Yaskawa INFORM job: BATMAN_NEW3.JBI

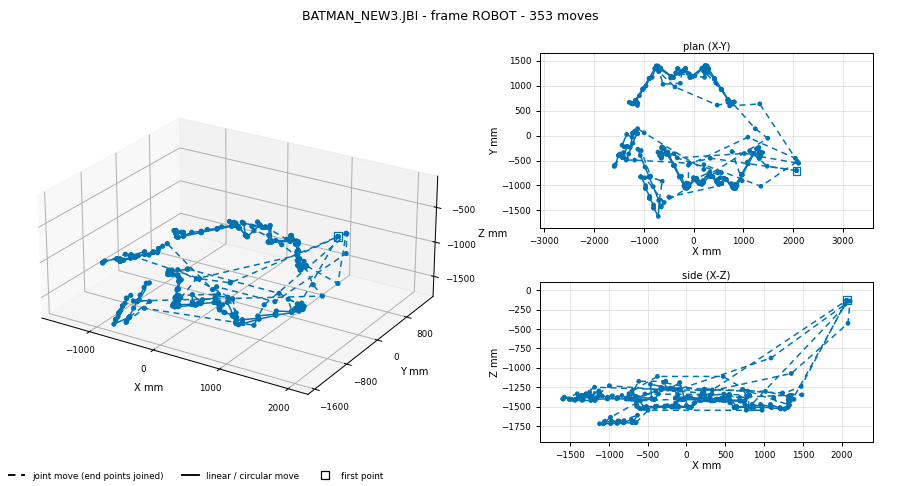
[picture p0: tool path of BATMAN_NEW3.JBI in frame ROBOT, 353 of 354 moves have a stored position in this frame; points joined in program order, loops and branches not executed]
/JOB
//NAME BATMAN_NEW3
//POS
///NPOS 437,437,353,19,0,1
///TOOL 0
///POSTYPE ROBOT
///RECTAN
///RCONF 0,0,0,0,0,0,0,0,0,0,0,0,0,0,0,0,0,0,0,0,0,0,0,0
C00000=2065.993,-701.065,-130.284,1.6748,-19.7957,-6.8086
C00001=2065.993,-701.066,-130.317,1.6736,-19.7947,-6.8065
C00002=1479.209,-614.254,-1239.827,11.6326,33.9671,-178.8219
C00003=1125.636,-307.051,-1381.425,11.6326,33.9683,179.6301
C00004=1211.356,-355.995,-1515.705,1.6711,33.5119,145.1887
C00005=1207.829,-356.009,-1519.032,1.6708,33.5119,145.1897
C00006=1207.807,-355.998,-1529.580,1.6710,33.5101,145.1899
C00007=1207.829,-356.009,-1519.032,1.6708,33.5119,145.1897
C00008=1226.216,-355.997,-1519.056,1.6724,33.5092,145.1902
C00009=1207.829,-356.009,-1519.032,1.6708,33.5119,145.1897
C00010=1082.252,-529.394,-1470.919,1.6706,33.5110,145.1945
C00011=1087.987,-562.193,-1501.828,1.6729,33.5117,145.1983
C00012=1088.014,-562.206,-1515.111,1.6726,33.5132,145.1983
C00013=1087.987,-562.193,-1501.828,1.6729,33.5117,145.1983
C00014=1116.737,-562.190,-1501.837,1.6716,33.5119,145.1949
C00015=1087.987,-562.193,-1501.828,1.6729,33.5117,145.1983
C00016=956.028,-780.276,-1470.920,1.6694,33.5121,145.1915
C00017=968.960,-788.125,-1498.527,1.6701,33.5115,145.1891
C00018=968.967,-788.120,-1508.943,1.6694,33.5115,145.1892
C00019=968.960,-788.125,-1498.527,1.6701,33.5115,145.1891
C00020=991.209,-788.123,-1498.543,1.6717,33.5108,145.1905
C00021=968.960,-788.125,-1498.527,1.6701,33.5115,145.1891
C00022=846.889,-978.207,-1470.921,1.6701,33.5116,145.1891
C00023=862.357,-1002.638,-1501.051,1.6670,33.5088,145.1850
C00024=862.345,-1002.624,-1509.122,1.6663,33.5074,145.1836
C00025=862.357,-1002.638,-1501.051,1.6670,33.5088,145.1850
C00026=878.170,-1002.616,-1501.076,1.6660,33.5090,145.1863
C00027=862.357,-1002.638,-1501.051,1.6670,33.5088,145.1850
C00028=751.878,-962.551,-1470.637,-9.9278,21.9341,47.3593
C00029=782.343,-1021.883,-1501.453,-6.5198,31.4589,38.6711
C00030=782.349,-1021.901,-1508.593,-6.5211,31.4595,38.6707
C00031=782.343,-1021.883,-1501.453,-6.5198,31.4589,38.6711
C00032=772.436,-1031.632,-1503.007,-6.5210,31.4603,38.6751
C00033=782.343,-1021.883,-1501.453,-6.5198,31.4589,38.6711
C00034=651.465,-878.509,-1502.529,-6.5193,31.4567,38.6726
C00035=649.681,-879.962,-1505.034,-6.5204,31.4570,38.6688
C00036=649.679,-879.971,-1512.967,-6.5216,31.4579,38.6721
C00037=649.681,-879.962,-1505.034,-6.5204,31.4570,38.6688
C00038=638.496,-885.487,-1507.904,-6.5213,31.4572,38.6690
C00039=649.681,-879.962,-1505.034,-6.5204,31.4570,38.6688
C00040=536.093,-844.110,-1358.224,-6.5194,31.4565,38.6698
C00041=485.208,-882.506,-1390.226,-6.5180,31.4566,38.6722
C00042=469.831,-925.588,-1412.310,-6.5196,31.4595,38.6720
C00043=469.838,-925.615,-1422.209,-6.5208,31.4607,38.6737
C00044=469.831,-925.588,-1412.310,-6.5196,31.4595,38.6720
C00045=460.916,-939.180,-1415.903,-6.5217,31.4610,38.6723
C00046=469.831,-925.588,-1412.310,-6.5196,31.4595,38.6720
C00047=390.944,-821.413,-1401.907,-6.5189,31.4593,38.6711
C00048=370.304,-823.702,-1415.949,-6.5184,31.4594,38.6679
C00049=370.309,-823.695,-1427.366,-6.5174,31.4589,38.6696
C00050=370.304,-823.702,-1415.949,-6.5184,31.4594,38.6679
C00051=362.481,-832.843,-1419.419,-6.5181,31.4591,38.6684
C00052=370.304,-823.702,-1415.949,-6.5184,31.4594,38.6679
C00053=304.377,-775.536,-1384.314,-6.5183,31.4594,38.6652
C00054=190.919,-901.974,-1384.308,6.6118,30.8401,128.8238
C00055=195.878,-934.762,-1411.685,6.6092,30.8405,128.8212
C00056=195.887,-934.767,-1420.325,6.6101,30.8407,128.8263
C00057=195.878,-934.762,-1411.685,6.6092,30.8405,128.8212
C00058=202.495,-948.084,-1414.851,6.6099,30.8403,128.8223
C00059=195.878,-934.762,-1411.685,6.6092,30.8405,128.8212
C00060=-1.386,-846.899,-1381.133,6.6069,30.8405,134.1399
C00061=-1.384,-846.902,-1485.292,6.6071,30.8406,134.1408
C00062=18.120,-884.199,-1503.049,6.6086,30.8410,134.1399
C00063=18.115,-884.194,-1511.506,6.6087,30.8409,134.1387
C00064=18.120,-884.199,-1503.049,6.6086,30.8410,134.1399
C00065=26.172,-895.008,-1505.663,6.6092,30.8415,134.1385
C00066=18.120,-884.199,-1503.049,6.6086,30.8410,134.1399
C00067=-111.813,-1001.782,-1489.786,6.6089,30.8396,134.1409
C00068=-110.516,-1020.985,-1499.218,6.6089,30.8402,134.1417
C00069=-110.523,-1020.998,-1507.131,6.6095,30.8409,134.1397
C00070=-110.516,-1020.985,-1499.218,6.6089,30.8402,134.1417
C00071=-104.498,-1031.543,-1502.310,6.6099,30.8394,134.1431
C00072=-110.516,-1020.985,-1499.218,6.6089,30.8402,134.1417
C00073=-134.961,-974.431,-1451.204,-0.2767,36.0814,31.9882
C00074=-184.395,-1006.620,-1494.709,-0.2788,36.0816,31.9875
C00075=-184.386,-1006.637,-1507.407,-0.2801,36.0816,31.9874
C00076=-184.395,-1006.620,-1494.709,-0.2788,36.0816,31.9875
C00077=-208.747,-1006.634,-1494.698,-0.2814,36.0810,31.9855
C00078=-184.395,-1006.620,-1494.709,-0.2788,36.0816,31.9875
C00079=-244.393,-814.940,-1486.725,-0.2795,36.0814,31.9846
C00080=-276.066,-822.621,-1495.047,-0.2812,36.0816,31.9820
C00081=-276.076,-822.621,-1505.407,-0.2803,36.0821,31.9829
C00082=-276.066,-822.621,-1495.047,-0.2812,36.0816,31.9820
C00083=-299.433,-822.605,-1495.065,-0.2798,36.0806,31.9846
C00084=-276.066,-822.621,-1495.047,-0.2812,36.0816,31.9820
C00085=-381.996,-597.063,-1495.018,-0.2830,36.0831,31.9834
C00086=-396.395,-597.055,-1498.231,-0.2823,36.0831,31.9838
C00087=-396.413,-597.067,-1510.313,-0.2821,36.0844,31.9835
C00088=-396.395,-597.055,-1498.231,-0.2823,36.0831,31.9838
C00089=-422.077,-597.035,-1498.242,-0.2815,36.0825,31.9834
C00090=-396.395,-597.055,-1498.231,-0.2823,36.0831,31.9838
C00091=-516.342,-329.683,-1498.242,-0.2858,36.0793,31.9791
C00092=-541.396,-335.433,-1515.036,-0.2853,36.0793,31.9798
C00093=-541.399,-335.427,-1525.902,-0.2848,36.0790,31.9796
C00094=-541.396,-335.433,-1515.036,-0.2853,36.0793,31.9798
C00095=-563.435,-335.446,-1515.016,-0.2858,36.0816,31.9782
C00096=-541.396,-335.433,-1515.036,-0.2853,36.0793,31.9798
C00097=-641.458,-364.123,-1372.142,-0.2839,36.0778,31.9819
C00098=-662.744,-397.701,-1394.268,-0.2832,36.0779,31.9810
C00099=-662.752,-397.694,-1404.858,-0.2824,36.0779,31.9809
C00100=-662.744,-397.701,-1394.268,-0.2832,36.0779,31.9810
C00101=-686.425,-397.683,-1394.265,-0.2810,36.0766,31.9839
C00102=-662.744,-397.701,-1394.268,-0.2832,36.0779,31.9810
C00103=-395.220,-362.676,-1299.812,-0.2837,36.0781,31.9812
C00104=-328.978,-445.538,-1251.827,-0.2820,36.0777,31.9846
C00105=1019.066,-358.271,-1303.588,-0.7093,36.3388,173.5111
C00106=1312.502,-388.638,-1368.088,-0.7090,36.3391,143.8761
C00107=1330.261,-409.263,-1395.611,-0.7097,36.3382,143.8752
C00108=1330.266,-409.258,-1408.665,-0.7105,36.3381,143.8742
C00109=1330.261,-409.263,-1395.611,-0.7097,36.3382,143.8752
C00110=1359.166,-409.282,-1395.624,-0.7081,36.3381,143.8755
C00111=1330.261,-409.263,-1395.611,-0.7097,36.3382,143.8752
C00112=1346.256,-330.236,-1377.208,-0.7085,36.3387,143.8760
C00113=1385.768,-339.505,-1405.683,-0.7074,36.3385,143.8819
C00114=1349.259,-407.967,-1405.698,-0.7099,36.3376,143.8723
C00115=1344.221,-409.875,-1407.374,-0.7109,36.3390,143.8722
C00116=1319.007,-459.412,-1408.358,-0.7127,36.3385,143.8707
C00117=1316.585,-457.113,-1411.355,-0.7151,36.3388,143.8640
C00118=1314.211,-431.828,-1419.878,-0.7170,36.3383,163.2059
C00119=1313.610,-343.846,-1457.563,-0.7163,36.3370,163.2057
C00120=1312.128,-239.426,-1504.329,-0.7192,36.3404,-169.8403
C00121=1302.531,-244.407,-1511.260,-0.7169,36.3409,-169.8377
C00122=1267.911,-263.148,-1529.181,-0.7174,36.3418,-169.8424
C00123=1265.622,-266.346,-1531.847,1.6688,33.5119,174.0846
C00124=1213.936,-359.434,-1529.128,7.9444,32.4168,142.7983
C00125=1097.826,-565.399,-1513.792,8.0761,31.8062,143.0840
C00126=978.992,-787.849,-1508.370,11.5262,32.2738,144.8308
C00127=870.875,-1002.933,-1509.595,7.8980,31.3909,142.8673
C00128=841.816,-1062.860,-1508.469,7.3802,28.2390,142.8982
C00129=553.926,-745.251,-1344.470,9.9580,22.3671,144.0884
C00130=553.926,-745.251,-1344.470,9.9580,22.3671,144.0884
C00131=-536.407,-379.228,-1337.930,-3.7346,30.6001,32.3556
C00132=-716.129,-331.806,-1403.803,-3.7368,30.5972,32.3471
C00133=-681.265,-398.771,-1403.765,-3.7327,30.5994,32.3525
C00134=-676.698,-399.723,-1405.572,-3.7330,30.6001,32.3555
C00135=-648.225,-452.003,-1403.979,-3.7329,30.5991,32.3574
C00136=-645.783,-446.417,-1409.426,-3.7316,30.5985,32.3594
C00137=-643.641,-424.031,-1414.162,6.8151,41.7178,38.5590
C00138=-642.472,-351.082,-1444.628,6.8142,41.7174,38.5597
C00139=-641.451,-256.638,-1485.774,6.7766,41.4625,22.9438
C00140=-638.655,-225.961,-1497.533,6.8201,41.7201,-9.7951
C00141=-606.472,-247.507,-1518.640,6.8237,41.7199,-9.7921
C00142=-589.700,-266.409,-1527.585,-3.7338,30.5952,1.6448
C00143=-548.411,-343.534,-1525.056,-3.7347,30.5964,37.9422
C00144=-403.963,-602.728,-1509.074,-3.7352,30.6012,40.7690
C00145=-284.220,-831.531,-1505.467,-3.7335,30.6016,39.5000
C00146=-193.310,-1012.463,-1505.473,-3.7341,30.5995,40.3635
C00147=-172.149,-1053.927,-1503.363,-3.7384,30.5988,41.1995
C00148=-143.820,-951.201,-1386.733,-3.7395,30.5979,32.3557
C00149=328.849,-733.445,-1337.611,2.7644,30.8890,70.6747
C00150=338.434,-799.747,-1424.588,2.7649,30.8868,70.6709
C00151=347.582,-809.529,-1424.840,2.7655,30.8869,70.6739
C00152=465.382,-936.963,-1420.390,2.7641,30.8894,70.6728
C00153=500.403,-974.854,-1419.495,2.7654,30.8881,70.6755
C00154=502.728,-975.948,-1420.152,2.7642,30.8887,70.6768
C00155=558.235,-964.171,-1445.639,29.9134,35.7054,85.7902
C00156=566.476,-953.294,-1452.395,19.5078,42.2162,79.2507
C00157=613.155,-854.018,-1511.422,19.5140,42.2128,79.2557
C00158=619.425,-859.852,-1512.190,3.7143,38.7707,68.9580
C00159=645.641,-886.484,-1510.742,-0.5875,30.5403,66.8343
C00160=773.682,-1027.269,-1508.152,1.6003,33.1198,67.9708
C00161=802.111,-1056.994,-1506.134,3.6680,32.7298,69.0087
C00162=802.122,-1056.982,-1354.174,6.2530,30.6739,70.3394
C00163=481.154,-746.898,-1337.541,6.2536,30.6743,70.3404
C00164=303.930,-769.190,-1354.154,12.5353,29.0330,117.3688
C00165=330.093,-802.167,-1423.714,12.5353,29.0320,117.3702
C00166=314.789,-820.264,-1426.190,12.5335,29.0340,117.3719
C00167=194.430,-949.182,-1419.608,12.5356,29.0341,117.3712
C00168=168.116,-977.659,-1418.609,12.5346,29.0295,117.3793
C00169=164.056,-975.884,-1418.609,12.5348,29.0312,117.3768
C00170=109.552,-964.850,-1447.287,-20.8943,38.2908,98.4122
C00171=97.137,-940.053,-1460.340,-8.8476,43.5866,106.1670
C00172=64.741,-867.815,-1502.677,-8.8482,43.5869,106.1635
C00173=57.160,-853.414,-1511.897,-8.8466,43.5860,106.1711
C00174=48.710,-862.514,-1512.138,-8.7696,29.7613,106.6801
C00175=-100.586,-1023.322,-1507.723,-8.7691,29.7615,106.6747
C00176=-133.949,-1058.932,-1505.596,-8.7707,29.7582,106.6747
C00177=-104.193,-961.904,-1408.358,-8.7704,29.7603,106.6778
C00178=-104.195,-589.697,-1279.272,-8.7711,29.7586,106.6768
C00179=1089.919,-31.439,-873.125,-36.7541,69.9873,137.0084
///RCONF 0,0,0,0,1,0,0,0,0,0,0,0,0,0,0,0,0,0,0,0,0,0,0,0
C00180=2042.728,-454.958,-183.433,1.6788,-19.8065,-6.7510
C00181=1329.047,637.602,-1479.857,8.0540,25.5528,30.8439
///RCONF 0,0,0,0,0,0,0,0,0,0,0,0,0,0,0,0,0,0,0,0,0,0,0,0
C00182=724.107,597.545,-1276.344,-3.2635,41.6684,-140.4024
C00183=785.383,659.459,-1372.820,-3.2632,41.6678,-140.4000
C00184=792.753,652.576,-1383.361,-3.2644,41.6697,-140.4060
C00185=785.383,659.459,-1372.820,-3.2632,41.6678,-140.4000
C00186=780.124,673.327,-1385.992,-3.2593,41.6675,-140.3923
C00187=785.383,659.459,-1372.820,-3.2632,41.6678,-140.4000
C00188=688.781,670.593,-1383.775,8.5921,32.7651,-134.9169
C00189=689.238,716.401,-1420.123,8.5921,32.7651,-134.9151
C00190=689.245,716.402,-1430.226,8.5926,32.7655,-134.9147
C00191=689.238,716.401,-1420.123,8.5921,32.7651,-134.9151
C00192=710.026,716.388,-1420.124,8.5932,32.7632,-134.9113
C00193=689.238,716.401,-1420.123,8.5921,32.7651,-134.9151
C00194=689.230,716.407,-1420.121,8.5916,32.7651,-134.9153
C00195=554.239,927.574,-1413.741,8.5900,32.7633,-134.9152
C00196=554.238,927.566,-1425.025,8.5905,32.7628,-134.9151
C00197=554.239,927.574,-1413.741,8.5900,32.7633,-134.9152
C00198=579.309,927.583,-1413.727,8.5909,32.7646,-134.9144
C00199=554.239,927.574,-1413.741,8.5900,32.7633,-134.9152
C00200=447.851,1057.003,-1392.108,8.5896,32.7630,-134.9175
C00201=417.599,1139.232,-1408.122,8.5926,32.7611,-134.9068
C00202=417.620,1139.241,-1415.890,8.5939,32.7624,-134.9057
C00203=417.599,1139.232,-1408.122,8.5926,32.7611,-134.9068
C00204=437.176,1139.232,-1408.121,8.5924,32.7608,-134.9064
C00205=417.599,1139.232,-1408.122,8.5926,32.7611,-134.9068
C00206=298.416,1271.074,-1391.633,8.5930,32.7623,-134.9078
C00207=293.017,1340.342,-1403.006,8.5942,32.7634,-134.9096
C00208=293.012,1340.335,-1412.621,8.5936,32.7630,-134.9120
C00209=293.017,1340.342,-1403.006,8.5942,32.7634,-134.9096
C00210=314.109,1340.332,-1403.005,8.5956,32.7645,-134.9108
C00211=293.017,1340.342,-1403.006,8.5942,32.7634,-134.9096
C00212=233.980,1302.281,-1344.762,8.5940,32.7640,-134.9075
C00213=200.134,1294.158,-1339.988,10.2608,31.0598,-45.0576
C00214=172.748,1341.866,-1398.059,10.2620,31.0622,-45.0581
C00215=172.750,1341.856,-1411.003,10.2608,31.0619,-45.0612
C00216=172.748,1341.866,-1398.059,10.2620,31.0622,-45.0581
C00217=162.053,1360.361,-1403.672,10.2607,31.0636,-45.0654
C00218=172.748,1341.866,-1398.059,10.2620,31.0622,-45.0581
C00219=26.821,1201.359,-1372.636,10.2610,31.0614,-45.0581
C00220=-26.114,1184.722,-1395.825,10.2614,31.0609,-45.0571
C00221=-26.119,1184.747,-1409.910,10.2622,31.0622,-45.0567
C00222=-26.114,1184.722,-1395.825,10.2614,31.0609,-45.0571
C00223=-38.557,1201.364,-1401.881,10.2611,31.0613,-45.0602
C00224=-26.114,1184.722,-1395.825,10.2614,31.0609,-45.0571
C00225=-85.944,1239.452,-1189.279,10.2632,31.0602,-45.0547
C00226=-202.376,1302.359,-1263.326,10.2654,31.0601,-39.0783
C00227=-202.377,1302.375,-1273.759,10.2665,31.0600,-39.0755
C00228=-202.376,1302.359,-1263.326,10.2654,31.0601,-39.0783
C00229=-213.401,1315.412,-1266.159,10.2653,31.0594,-39.0754
C00230=-202.376,1302.359,-1263.326,10.2654,31.0601,-39.0783
C00231=-463.805,1156.888,-1211.984,5.4408,32.3182,-121.2144
C00232=-448.455,1180.872,-1396.312,5.4420,32.3182,-121.2130
C00233=-448.461,1180.875,-1405.887,5.4414,32.3181,-121.2136
C00234=-448.455,1180.872,-1396.312,5.4420,32.3182,-121.2130
C00235=-438.739,1194.365,-1399.533,5.4424,32.3182,-121.2152
C00236=-448.455,1180.872,-1396.312,5.4420,32.3182,-121.2130
C00237=-657.730,1329.361,-1367.973,5.4433,32.3188,-121.2093
C00238=-663.299,1347.249,-1396.310,5.4469,32.3207,-121.2088
C00239=-663.288,1347.263,-1404.262,5.4479,32.3220,-121.2052
C00240=-663.299,1347.249,-1396.310,5.4469,32.3207,-121.2088
C00241=-654.469,1361.022,-1397.928,5.4472,32.3207,-121.2069
C00242=-663.299,1347.249,-1396.310,5.4469,32.3207,-121.2088
C00243=-698.479,1323.579,-1333.586,5.4477,32.3218,-121.2085
C00244=-740.743,1333.011,-1333.582,5.4466,32.3224,-21.5902
C00245=-770.855,1345.163,-1390.229,5.4461,32.3244,-21.5929
C00246=-770.847,1345.152,-1402.397,5.4455,32.3237,-21.5937
C00247=-770.855,1345.163,-1390.229,5.4461,32.3244,-21.5929
C00248=-795.277,1345.162,-1390.244,5.4458,32.3245,-21.5940
C00249=-770.855,1345.163,-1390.229,5.4461,32.3244,-21.5929
C00250=-831.818,1170.618,-1356.598,5.4477,32.3246,-21.5912
C00251=-886.559,1145.436,-1385.426,5.4460,32.3239,-21.5899
C00252=-886.565,1145.436,-1399.683,5.4454,32.3246,-21.5914
C00253=-886.559,1145.436,-1385.426,5.4460,32.3239,-21.5899
C00254=-917.367,1145.449,-1385.412,5.4486,32.3247,-21.5896
C00255=-886.559,1145.436,-1385.426,5.4460,32.3239,-21.5899
C00256=-956.142,996.150,-1360.002,5.4455,32.3233,-21.5898
C00257=-1015.444,934.058,-1379.897,5.4455,32.3192,-21.5922
C00258=-1015.421,934.048,-1400.561,5.4457,32.3177,-21.5921
C00259=-1015.437,934.045,-1399.064,5.4450,32.3186,-21.5914
C00260=-1015.444,934.058,-1379.897,5.4455,32.3192,-21.5922
C00261=-1051.411,934.058,-1379.898,5.4445,32.3193,-21.5956
C00262=-1015.444,934.058,-1379.897,5.4455,32.3192,-21.5922
C00263=-1086.808,802.572,-1361.725,5.4423,32.3202,-21.5974
C00264=-1159.323,707.147,-1394.101,5.4407,32.3217,-21.6008
C00265=-1159.296,707.145,-1406.974,5.4389,32.3209,-21.6105
C00266=-1159.323,707.147,-1394.101,5.4407,32.3217,-21.6008
C00267=-1187.279,707.135,-1394.079,5.4396,32.3232,-21.5966
C00268=-1159.323,707.147,-1394.101,5.4407,32.3217,-21.6008
C00269=-1128.608,606.997,-1296.811,5.4402,32.3220,-21.6018
C00270=-1245.560,650.345,-1363.191,5.4391,32.3216,-21.6043
C00271=-1253.840,659.612,-1369.532,5.4396,32.3086,-21.6048
C00272=-1245.560,650.345,-1363.191,5.4391,32.3216,-21.6043
C00273=-1255.518,641.298,-1375.299,5.4388,32.3217,-21.6053
C00274=-1245.560,650.345,-1363.191,5.4391,32.3216,-21.6043
C00275=-1122.499,650.360,-1312.804,5.4384,32.3212,-21.6061
C00276=-1246.019,650.333,-1312.805,-5.9814,50.4641,-44.8970
C00277=-1292.164,668.745,-1333.265,-5.9790,50.4644,-44.8908
C00278=-1231.709,639.662,-1400.187,-5.9769,50.4666,-44.8863
C00279=-1218.432,639.336,-1404.695,9.2051,37.0994,-34.2739
C00280=-1209.403,648.076,-1408.638,9.2048,37.0993,-34.2731
C00281=-1170.360,710.291,-1406.670,9.2055,37.0992,-34.2737
C00282=-1024.371,936.002,-1398.258,9.2078,37.1003,-34.2692
C00283=-896.601,1150.196,-1398.253,9.2032,37.1000,-34.2694
C00284=-781.119,1345.938,-1400.544,9.2147,37.0957,-34.2682
C00285=-750.870,1396.710,-1400.505,9.2146,37.0994,-34.2694
C00286=-748.321,1400.053,-1400.515,9.2140,37.0989,-34.2683
C00287=-701.755,1284.519,-1299.250,9.2134,37.0978,-34.2698
C00288=-374.253,977.072,-1110.582,-16.3615,18.9747,-168.4330
C00289=472.792,614.034,-1110.590,-6.3310,51.0848,-162.4334
C00290=790.077,666.826,-1299.714,-6.3326,51.0845,-162.4374
C00291=816.173,675.910,-1358.543,-6.3341,51.0842,-155.2649
C00292=816.177,676.401,-1355.243,-6.3377,51.0852,-155.2687
C00293=757.587,649.690,-1417.955,-6.3357,51.0871,-155.2635
C00294=745.147,646.476,-1430.103,-12.0666,41.5969,-159.4258
C00295=739.613,652.892,-1430.747,-14.7082,35.8520,-158.3156
C00296=698.688,719.019,-1430.343,-14.7066,35.8512,-158.3093
C00297=562.776,933.439,-1425.541,-14.7084,35.8506,-158.3083
C00298=425.344,1144.525,-1415.822,-14.7098,35.8488,-158.3129
C00299=301.450,1344.182,-1413.742,-14.7101,35.8478,-158.3119
C00300=272.598,1391.057,-1413.172,-14.7077,35.8494,-158.3072
C00301=260.911,1405.768,-1411.522,-14.7076,35.8478,-158.3086
C00302=220.093,1170.732,-1299.028,-14.7077,35.8474,-158.3065
C00303=-294.154,1247.220,-1186.692,-14.7086,35.8481,-158.3060
C00304=-242.562,1288.482,-1273.150,-14.2330,35.5827,-141.3920
C00305=-312.356,1343.179,-1273.798,-14.2228,35.5979,-141.3866
C00306=-318.403,1347.498,-1273.796,-14.2220,35.5979,-141.3873
C00307=-322.718,1340.149,-1279.722,-14.2217,35.5982,-157.9762
C00308=-360.883,1261.425,-1337.016,-14.2215,35.5979,-157.9820
C00309=-406.935,1168.469,-1402.157,-14.2214,35.5994,-157.9829
C00310=-409.683,1164.442,-1406.283,-14.2227,35.5996,-147.9815
C00311=-417.765,1170.563,-1406.551,-14.2208,35.6000,-147.9803
C00312=-440.479,1187.915,-1406.121,-14.2208,35.6025,-144.4920
C00313=-660.238,1358.264,-1403.716,-14.2203,35.6056,-144.4919
C00314=-713.517,1398.596,-1402.095,-14.2235,35.6053,-144.4993
C00315=-702.785,1334.590,-1330.560,-14.2225,35.6052,-144.4992
C00316=-615.113,1031.882,-1174.072,-14.2237,35.6047,-144.5023
C00317=-266.790,1052.428,-1172.785,14.1594,35.6599,-52.4229
C00318=-234.621,1290.298,-1271.352,14.1573,35.6533,-52.4193
C00319=-170.266,1343.198,-1274.471,14.1621,35.6578,-52.4205
C00320=-163.350,1347.913,-1274.487,14.1614,35.6572,-52.4200
C00321=-161.403,1342.862,-1281.279,7.3802,43.3671,-41.1599
C00322=-113.870,1250.739,-1345.243,7.3795,43.3689,-41.1646
C00323=-75.578,1173.045,-1403.534,7.3827,43.3703,-41.1594
C00324=-71.378,1165.451,-1408.302,7.3856,43.3696,-41.1548
C00325=-59.197,1175.793,-1409.651,4.6384,38.1537,-42.8411
C00326=-35.448,1195.776,-1410.312,4.6465,38.1543,-47.5801
C00327=166.563,1354.922,-1410.948,4.6441,38.1493,-47.5848
C00328=227.339,1402.932,-1410.926,4.6442,38.1483,-47.5854
C00329=233.128,1408.173,-1410.916,4.6445,38.1490,-47.5846
C00330=233.146,1258.590,-1276.348,4.6463,38.1495,-47.5846
C00331=233.273,1258.338,-1276.378,4.6470,38.1496,-47.5838
C00332=233.273,1258.338,-1276.378,4.6470,38.1496,-47.5838
C00333=233.248,1273.531,-1276.386,4.6460,38.1499,-47.5825
C00334=1238.436,139.129,-1323.509,-1.5927,36.9682,-135.2428
C00335=1488.778,-52.476,-1347.695,27.2487,24.5669,-70.7938
C00336=-591.325,-1341.846,-1422.510,-0.6043,40.8297,16.7434
C00337=-978.344,-845.186,-1637.203,-0.6000,40.8277,16.7477
C00338=-1060.712,-827.560,-1707.784,-0.5964,40.8264,16.7530
C00339=-1060.716,-827.565,-1719.613,-0.5979,40.8266,16.7496
C00340=-1060.712,-827.560,-1707.784,-0.5964,40.8264,16.7530
C00341=-1076.749,-827.566,-1707.781,-0.5968,40.8274,16.7526
C00342=-1060.712,-827.560,-1707.784,-0.5964,40.8264,16.7530
C00343=-964.064,-1003.361,-1685.365,-0.5978,40.8280,16.7499
C00344=-967.258,-1055.832,-1705.053,-0.5976,40.8279,16.7488
C00345=-967.265,-1055.827,-1717.171,-0.5974,40.8281,16.7474
C00346=-967.258,-1055.832,-1705.053,-0.5976,40.8279,16.7488
C00347=-984.967,-1055.847,-1705.045,-0.5977,40.8287,16.7479
C00348=-967.258,-1055.832,-1705.053,-0.5976,40.8279,16.7488
C00349=-883.106,-1217.890,-1684.422,-0.5980,40.8275,16.7460
C00350=-884.555,-1256.605,-1703.312,-0.5986,40.8276,16.7466
C00351=-884.543,-1256.571,-1713.321,-0.5947,40.8260,16.7508
C00352=-884.555,-1256.605,-1703.312,-0.5986,40.8276,16.7466
C00353=-901.563,-1256.594,-1703.316,-0.6002,40.8264,16.7423
C00354=-884.555,-1256.605,-1703.312,-0.5986,40.8276,16.7466
C00355=-804.394,-1392.262,-1680.447,-0.5972,40.8269,16.7457
C00356=-802.318,-1451.144,-1699.808,-0.5973,40.8272,16.7464
C00357=-802.295,-1451.144,-1709.722,-0.5981,40.8252,16.7458
C00358=-802.318,-1451.144,-1699.808,-0.5973,40.8272,16.7464
C00359=-820.040,-1451.129,-1699.830,-0.5958,40.8269,16.7480
C00360=-802.318,-1451.144,-1699.808,-0.5973,40.8272,16.7464
C00361=-709.611,-1620.676,-1670.338,-0.5978,40.8273,16.7476
C00362=-689.604,-1294.748,-1695.996,-0.5975,40.8268,16.7459
C00363=-689.614,-1294.765,-1707.440,-0.5999,40.8277,16.7418
C00364=-689.604,-1294.748,-1695.996,-0.5975,40.8268,16.7459
C00365=-710.807,-1294.753,-1696.008,-0.5986,40.8259,16.7454
C00366=-689.604,-1294.748,-1695.996,-0.5975,40.8268,16.7459
C00367=-630.511,-916.030,-1610.753,-0.6017,40.8266,16.7401
C00368=-868.430,-829.435,-1692.124,-0.6028,40.8258,16.7353
C00369=-892.870,-831.979,-1714.985,-0.5981,40.8255,16.7444
C00370=-976.713,-630.080,-1718.549,-0.6011,40.8246,16.7412
C00371=-1071.217,-398.415,-1720.690,-0.6000,40.8208,16.7397
C00372=-1119.996,-273.264,-1720.027,-0.6007,40.8208,16.7405
C00373=-1052.650,-299.020,-1688.341,-0.6009,40.8211,16.7408
C00374=-865.284,-812.787,-1688.334,-0.6039,40.8202,42.9608
C00375=-892.749,-830.002,-1713.253,-0.5986,40.8166,42.9666
C00376=-812.172,-1024.012,-1709.563,-0.6014,40.8165,42.9567
C00377=-700.538,-1299.832,-1707.155,-0.6008,40.8192,42.9610
C00378=-657.041,-1411.182,-1706.542,-0.5992,40.8178,42.9644
C00379=-649.131,-1432.542,-1706.544,-0.5977,40.8180,42.9663
C00380=-495.179,-1232.483,-1546.245,-0.5800,40.8231,42.9777
C00381=975.318,-905.329,-1546.300,2.7447,40.6858,121.3068
C00382=771.357,-320.253,-1546.238,-0.5794,40.8236,124.0583
///RCONF 0,0,0,0,1,0,0,0,0,0,0,0,0,0,0,0,0,0,0,0,0,0,0,0
C00383=2108.910,-555.323,-138.194,2.1712,-19.6918,-3.5371
///RCONF 0,0,0,0,0,0,0,0,0,0,0,0,0,0,0,0,0,0,0,0,0,0,0,0
C00384=2082.559,-517.688,-426.187,17.7899,-11.9984,-30.1124
C00385=1351.715,-1016.627,-1072.730,14.7650,1.4143,-53.7135
C00386=205.703,-583.482,-1322.085,9.2825,24.4184,-95.9833
C00387=203.961,-679.195,-1324.426,-9.5613,21.9567,95.9050
C00388=-993.168,56.729,-1229.540,-0.2104,49.9239,-21.9207
C00389=-1124.976,139.813,-1330.335,5.3125,39.0598,-25.3648
C00390=-1217.958,48.598,-1401.440,5.3913,38.9364,-25.3168
C00391=-1222.465,48.743,-1409.263,5.3874,38.9378,-25.3223
C00392=-1222.459,48.730,-1420.612,5.3858,38.9371,-25.3242
C00393=-1222.465,48.743,-1409.263,5.3874,38.9378,-25.3223
C00394=-1239.080,48.748,-1409.236,5.3856,38.9399,-25.3266
C00395=-1222.465,48.743,-1409.263,5.3874,38.9378,-25.3223
C00396=-1271.414,-233.653,-1365.903,5.3880,38.9368,-25.3214
C00397=-1335.102,-218.968,-1407.739,5.3747,38.9270,-25.3244
C00398=-1335.110,-218.964,-1419.095,5.3738,38.9278,-25.3274
C00399=-1335.102,-218.968,-1407.739,5.3747,38.9270,-25.3244
C00400=-1351.938,-218.955,-1407.734,5.3749,38.9273,-25.3233
C00401=-1335.102,-218.968,-1407.739,5.3747,38.9270,-25.3244
C00402=-1410.796,-411.626,-1397.644,5.3751,38.9281,-25.3225
C00403=-1428.227,-437.232,-1406.270,5.3763,38.9287,-25.3214
C00404=-1428.230,-437.231,-1419.122,5.3758,38.9290,-25.3227
C00405=-1428.227,-437.232,-1406.270,5.3763,38.9287,-25.3214
C00406=-1445.183,-437.215,-1406.274,5.3770,38.9284,-25.3233
C00407=-1428.227,-437.232,-1406.270,5.3763,38.9287,-25.3214
C00408=-1478.764,-369.056,-1406.265,5.3746,38.9285,-25.3278
C00409=-1508.274,-399.507,-1403.549,5.3752,38.9282,-25.3298
C00410=-1508.284,-399.505,-1415.860,5.3764,38.9286,-25.3265
C00411=-1508.274,-399.507,-1403.549,5.3752,38.9282,-25.3298
C00412=-1525.499,-399.503,-1403.534,5.3741,38.9288,-25.3312
C00413=-1508.274,-399.507,-1403.549,5.3752,38.9282,-25.3298
C00414=-1573.700,-586.702,-1378.129,5.3749,38.9274,-25.3303
C00415=-1591.625,-610.872,-1399.727,5.3751,38.9284,-25.3300
C00416=-1591.607,-610.857,-1410.848,5.3774,38.9278,-25.3276
C00417=-1591.625,-610.872,-1399.727,5.3751,38.9284,-25.3300
C00418=-1607.585,-610.886,-1399.726,5.3748,38.9284,-25.3293
C00419=-1591.625,-610.872,-1399.727,5.3751,38.9284,-25.3300
C00420=-1407.614,-340.295,-1334.283,5.3763,38.9277,-25.3283
C00421=-1393.545,-225.421,-1380.034,5.3755,38.9268,-25.3271
C00422=-1436.319,-192.923,-1419.519,-0.6441,37.4048,-43.4681
C00423=-1343.970,24.204,-1419.685,-0.6458,37.4045,-43.4729
C00424=-1233.172,-33.364,-1421.676,-0.6450,37.4042,-43.4706
C00425=-1180.498,93.004,-1421.467,-0.6445,37.4051,-43.4715
C00426=-1123.867,39.567,-1327.748,-0.6454,37.4059,-43.4725
C00427=-1123.867,39.567,-1327.748,-0.6454,37.4059,-43.4725
C00428=-1139.614,46.545,-1367.957,-0.6485,37.4091,-15.9314
C00429=-1221.149,-154.590,-1364.989,-0.6505,37.4071,-15.9367
C00430=-1304.293,-367.690,-1359.056,-0.6521,37.4085,-15.9430
C00431=-1343.286,-469.596,-1355.805,-0.6535,37.4062,-15.9492
C00432=-1354.672,-491.189,-1354.002,-0.6534,37.4048,-15.9508
C00433=-1184.082,-491.180,-1249.860,-0.6521,37.4040,-15.9519
C00434=-78.969,-554.378,-1286.716,1.4249,23.3229,2.1506
C00435=333.912,-453.248,-1285.762,1.2790,23.3311,46.5433
C00436=2065.993,-701.065,-130.284,1.6748,-19.7957,-6.8086
BC00000=430.297,4179.635,1999.619
BC00001=506.026,2934.354,1999.615
BC00002=506.026,2197.799,889.024
BC00003=1028.979,2071.524,879.911
BC00004=1028.979,2071.524,879.911
BC00005=1028.979,2071.524,879.911
BC00006=1028.979,2071.524,879.911
BC00007=1028.979,2071.524,879.911
BC00008=1028.979,2071.524,879.911
BC00009=1028.979,2071.524,879.911
BC00010=1028.973,2071.524,879.905
BC00011=1028.973,2071.524,879.905
BC00012=1028.973,2071.524,879.905
BC00013=1028.973,2071.524,879.905
BC00014=1028.973,2071.524,879.905
BC00015=1028.973,2071.524,879.905
BC00016=1028.973,2071.524,879.905
BC00017=1028.973,2071.524,879.905
BC00018=1028.973,2071.524,879.905
BC00019=1028.973,2071.524,879.905
BC00020=1028.973,2071.524,879.905
BC00021=1028.973,2071.524,879.905
BC00022=1028.973,2071.524,879.905
BC00023=1028.973,2071.524,879.905
BC00024=1028.973,2071.524,879.905
BC00025=1028.973,2071.524,879.905
BC00026=1028.973,2071.524,879.905
BC00027=1028.973,2071.524,879.905
BC00028=1028.973,2071.524,879.905
BC00029=1028.973,2071.524,879.905
BC00030=1028.973,2071.524,879.905
BC00031=1028.973,2071.524,879.905
BC00032=1028.973,2071.524,879.905
BC00033=1028.973,2071.524,879.905
BC00034=1028.973,2071.524,879.905
BC00035=1028.973,2071.524,879.905
BC00036=1028.973,2071.524,879.905
BC00037=1028.973,2071.524,879.905
BC00038=1028.973,2071.524,879.905
BC00039=1028.973,2071.524,879.905
BC00040=1028.973,2071.524,879.905
BC00041=1028.973,2071.524,879.905
BC00042=1028.973,2071.524,879.905
BC00043=1028.973,2071.524,879.905
BC00044=1028.973,2071.524,879.905
BC00045=1028.973,2071.524,879.905
BC00046=1028.973,2071.524,879.905
BC00047=1028.973,2071.524,879.905
BC00048=1028.973,2071.524,879.905
BC00049=1028.973,2071.524,879.905
BC00050=1028.973,2071.524,879.905
BC00051=1028.973,2071.524,879.905
BC00052=1028.973,2071.524,879.905
BC00053=1028.973,2071.524,879.905
BC00054=1028.973,2071.524,879.905
BC00055=1028.973,2071.524,879.905
BC00056=1028.973,2071.524,879.905
BC00057=1028.973,2071.524,879.905
BC00058=1028.973,2071.524,879.905
BC00059=1028.973,2071.524,879.905
BC00060=1028.973,2071.524,879.905
BC00061=1028.973,2071.524,879.905
BC00062=1028.973,2071.524,879.905
BC00063=1028.973,2071.524,879.905
BC00064=1028.973,2071.524,879.905
BC00065=1028.973,2071.524,879.905
BC00066=1028.973,2071.524,879.905
BC00067=1028.973,2071.524,879.905
BC00068=1028.973,2071.524,879.905
BC00069=1028.973,2071.524,879.905
BC00070=1028.973,2071.524,879.905
BC00071=1028.973,2071.524,879.905
BC00072=1028.973,2071.524,879.905
BC00073=1028.973,2071.524,879.905
BC00074=1028.973,2071.524,879.905
BC00075=1028.973,2071.524,879.905
BC00076=1028.973,2071.524,879.905
BC00077=1028.973,2071.524,879.905
BC00078=1028.973,2071.524,879.905
BC00079=1028.973,2071.524,879.905
BC00080=1028.973,2071.524,879.905
BC00081=1028.973,2071.524,879.905
BC00082=1028.973,2071.524,879.905
BC00083=1028.973,2071.524,879.905
BC00084=1028.973,2071.524,879.905
BC00085=1028.973,2071.524,879.905
BC00086=1028.973,2071.524,879.905
BC00087=1028.973,2071.524,879.905
BC00088=1028.973,2071.524,879.905
BC00089=1028.973,2071.524,879.905
BC00090=1028.973,2071.524,879.905
BC00091=1028.973,2071.524,879.905
BC00092=1028.973,2071.524,879.905
BC00093=1028.973,2071.524,879.905
BC00094=1028.973,2071.524,879.905
BC00095=1028.973,2071.524,879.905
BC00096=1028.973,2071.524,879.905
BC00097=1028.973,2071.524,879.905
BC00098=1028.973,2071.524,879.905
BC00099=1028.973,2071.524,879.905
BC00100=1028.973,2071.524,879.905
BC00101=1028.973,2071.524,879.905
BC00102=1028.973,2071.524,879.905
BC00103=1028.973,2071.524,879.905
BC00104=1028.973,2071.524,879.905
BC00105=1028.973,2071.524,879.905
BC00106=1028.973,2071.524,879.905
BC00107=1028.973,2071.524,879.905
BC00108=1028.973,2071.524,879.905
BC00109=1028.973,2071.524,879.905
BC00110=1028.973,2071.524,879.905
BC00111=1028.973,2071.524,879.905
BC00112=1028.973,2071.524,879.905
BC00113=1028.973,2071.524,879.905
BC00114=1028.973,2071.524,879.905
BC00115=1028.973,2071.524,879.905
BC00116=1028.973,2071.524,879.905
BC00117=1028.973,2071.524,879.905
BC00118=1028.973,2071.524,879.905
BC00119=1028.973,2071.524,879.905
BC00120=1028.973,2071.524,879.905
BC00121=1028.973,2071.524,879.905
BC00122=1028.973,2071.524,879.905
BC00123=1028.979,2071.524,879.911
BC00124=1028.979,2071.524,879.911
BC00125=1028.979,2071.524,879.911
BC00126=1028.979,2071.524,879.911
BC00127=1028.979,2071.524,879.911
BC00128=1028.979,2071.524,879.911
BC00129=1028.979,2071.531,879.905
BC00130=1028.979,2071.531,1132.335
BC00131=1028.979,2071.531,879.905
BC00132=1028.979,2071.531,879.905
BC00133=1028.979,2071.531,879.905
BC00134=1028.979,2071.531,879.905
BC00135=1028.979,2071.531,879.905
BC00136=1028.979,2071.531,879.905
BC00137=1028.979,2071.531,879.905
BC00138=1028.979,2071.531,879.905
BC00139=1028.979,2071.531,879.905
BC00140=1028.979,2071.531,879.905
BC00141=1028.979,2071.531,879.905
BC00142=1028.979,2071.531,879.905
BC00143=1028.979,2071.531,879.905
BC00144=1028.979,2071.531,879.905
BC00145=1028.979,2071.531,879.905
BC00146=1028.979,2071.531,879.905
BC00147=1028.979,2071.531,879.905
BC00148=1028.979,2071.531,879.905
BC00149=1028.979,2071.531,879.905
BC00150=1028.979,2071.531,879.905
BC00151=1028.979,2071.531,879.905
BC00152=1028.979,2071.531,879.905
BC00153=1028.979,2071.531,879.905
BC00154=1028.979,2071.531,879.905
BC00155=1028.979,2071.531,879.905
BC00156=1028.979,2071.531,879.905
BC00157=1028.979,2071.531,879.905
BC00158=1028.979,2071.531,879.905
BC00159=1028.973,2071.537,879.898
BC00160=1028.979,2071.531,879.905
BC00161=1028.979,2071.531,879.905
BC00162=1028.979,2071.531,879.905
BC00163=1028.979,2071.531,879.905
BC00164=1028.979,2071.531,879.905
BC00165=1028.979,2071.531,879.905
BC00166=1028.979,2071.531,879.905
BC00167=1028.979,2071.531,879.905
BC00168=1028.979,2071.531,879.905
BC00169=1028.979,2071.531,879.905
BC00170=1028.979,2071.531,879.905
BC00171=1028.979,2071.531,879.905
BC00172=1028.979,2071.531,879.905
BC00173=1028.979,2071.531,879.905
BC00174=1028.979,2071.531,879.905
BC00175=1028.979,2071.531,879.905
BC00176=1028.979,2071.531,879.905
BC00177=1028.979,2071.531,879.905
BC00178=1028.979,2071.531,1313.400
BC00179=705.175,35.017,1952.866
BC00180=786.422,38.780,1999.645
BC00181=786.422,38.780,1999.645
BC00182=1602.623,32.856,1148.414
BC00183=1602.623,32.856,1148.414
BC00184=1602.623,32.856,1148.414
BC00185=1602.623,32.856,1148.414
BC00186=1602.623,32.856,1148.414
BC00187=1602.623,32.856,1148.414
BC00188=1602.623,32.856,1148.414
BC00189=1602.623,32.856,1148.414
BC00190=1602.623,32.856,1148.414
BC00191=1602.623,32.856,1148.414
BC00192=1602.623,32.856,1148.414
BC00193=1602.623,32.856,1148.414
BC00194=1602.623,32.856,1148.414
BC00195=1602.623,32.856,1148.414
BC00196=1602.623,32.856,1148.414
BC00197=1602.623,32.856,1148.414
BC00198=1602.623,32.856,1148.414
BC00199=1602.623,32.856,1148.414
BC00200=1602.623,32.856,1148.414
BC00201=1602.623,32.856,1148.414
BC00202=1602.623,32.856,1148.414
BC00203=1602.623,32.856,1148.414
BC00204=1602.623,32.856,1148.414
BC00205=1602.623,32.856,1148.414
BC00206=1602.623,32.856,1148.414
BC00207=1602.623,32.856,1148.414
BC00208=1602.623,32.856,1148.414
BC00209=1602.623,32.856,1148.414
BC00210=1602.623,32.856,1148.414
BC00211=1602.623,32.856,1148.414
BC00212=1602.623,32.856,1148.414
BC00213=1602.623,32.856,1148.414
BC00214=1602.623,32.856,1148.414
BC00215=1602.623,32.856,1148.414
BC00216=1602.623,32.856,1148.414
BC00217=1602.623,32.856,1148.414
BC00218=1602.623,32.856,1148.414
BC00219=1602.623,32.856,1148.414
BC00220=1602.623,32.856,1148.414
BC00221=1602.623,32.856,1148.414
BC00222=1602.623,32.856,1148.414
BC00223=1602.623,32.856,1148.414
BC00224=1602.623,32.856,1148.414
BC00225=1602.623,32.856,1148.414
BC00226=1602.623,32.856,1148.414
BC00227=1602.623,32.856,1148.414
BC00228=1602.623,32.856,1148.414
BC00229=1602.623,32.856,1148.414
BC00230=1602.623,32.856,1148.414
BC00231=1602.623,32.856,1148.414
BC00232=1602.623,32.856,1148.414
BC00233=1602.623,32.856,1148.414
BC00234=1602.623,32.856,1148.414
BC00235=1602.623,32.856,1148.414
BC00236=1602.623,32.856,1148.414
BC00237=1602.623,32.856,1148.414
BC00238=1602.623,32.856,1148.414
BC00239=1602.623,32.856,1148.414
BC00240=1602.623,32.856,1148.414
BC00241=1602.623,32.856,1148.414
BC00242=1602.623,32.856,1148.414
BC00243=1602.623,32.856,1148.414
BC00244=1602.623,32.856,1148.414
BC00245=1602.623,32.856,1148.414
BC00246=1602.623,32.856,1148.414
BC00247=1602.623,32.856,1148.414
BC00248=1602.623,32.856,1148.414
BC00249=1602.623,32.856,1148.414
BC00250=1602.623,32.856,1148.414
BC00251=1602.623,32.856,1148.414
BC00252=1602.623,32.856,1148.414
BC00253=1602.623,32.856,1148.414
BC00254=1602.623,32.856,1148.414
BC00255=1602.623,32.856,1148.414
BC00256=1602.623,32.856,1148.414
BC00257=1602.623,32.856,1148.414
BC00258=1602.623,32.856,1148.414
BC00259=1602.623,32.856,1148.414
BC00260=1602.623,32.856,1148.414
BC00261=1602.623,32.856,1148.414
BC00262=1602.623,32.856,1148.414
BC00263=1602.623,32.856,1148.414
BC00264=1602.623,32.856,1148.414
BC00265=1602.623,32.856,1148.414
BC00266=1602.623,32.856,1148.414
BC00267=1602.623,32.856,1148.414
BC00268=1602.623,32.856,1148.414
BC00269=1602.623,32.856,1148.414
BC00270=1602.623,32.856,1148.414
BC00271=1602.617,32.863,1148.408
BC00272=1602.623,32.856,1148.414
BC00273=1602.623,32.856,1148.414
BC00274=1602.623,32.856,1148.414
BC00275=1602.623,32.856,1148.414
BC00276=1602.623,32.856,1148.414
BC00277=1602.623,32.856,1148.414
BC00278=1602.623,32.856,1148.414
BC00279=1602.623,32.856,1148.414
BC00280=1602.623,32.856,1148.414
BC00281=1602.623,32.856,1148.414
BC00282=1602.623,32.856,1148.414
BC00283=1602.623,32.856,1148.414
BC00284=1602.617,32.856,1148.408
BC00285=1602.617,32.856,1148.408
BC00286=1602.617,32.856,1148.408
BC00287=1602.617,32.856,1148.408
BC00288=1602.617,32.856,1148.408
BC00289=1602.617,32.856,1148.408
BC00290=1602.617,32.856,1148.408
BC00291=1602.617,32.856,1148.408
BC00292=1602.610,32.863,1148.395
BC00293=1602.610,32.863,1148.395
BC00294=1602.610,32.863,1148.395
BC00295=1602.610,32.863,1148.395
BC00296=1602.610,32.863,1148.395
BC00297=1602.610,32.863,1148.395
BC00298=1602.610,32.863,1148.395
BC00299=1602.610,32.863,1148.395
BC00300=1602.610,32.863,1148.395
BC00301=1602.610,32.863,1148.395
BC00302=1602.610,32.863,1148.395
BC00303=1602.610,32.863,1148.395
BC00304=1602.610,32.863,1148.395
BC00305=1602.610,32.863,1148.391
BC00306=1602.610,32.863,1148.391
BC00307=1602.610,32.863,1148.391
BC00308=1602.610,32.863,1148.391
BC00309=1602.610,32.863,1148.391
BC00310=1602.610,32.863,1148.391
BC00311=1602.610,32.863,1148.391
BC00312=1602.610,32.863,1148.391
BC00313=1602.610,32.863,1148.391
BC00314=1602.610,32.863,1148.391
BC00315=1602.610,32.863,1148.391
BC00316=1602.610,32.863,1148.391
BC00317=1602.610,32.863,1148.391
BC00318=1602.617,32.863,1148.387
BC00319=1602.617,32.863,1148.387
BC00320=1602.617,32.863,1148.387
BC00321=1602.617,32.863,1148.387
BC00322=1602.617,32.863,1148.387
BC00323=1602.617,32.863,1148.387
BC00324=1602.617,32.863,1148.387
BC00325=1602.617,32.863,1148.387
BC00326=1602.617,32.863,1148.387
BC00327=1602.617,32.863,1148.387
BC00328=1602.617,32.863,1148.387
BC00329=1602.617,32.863,1148.387
BC00330=1602.617,32.863,1148.387
BC00331=1602.617,32.863,1960.335
BC00332=2287.550,32.863,1960.335
BC00333=2172.832,3214.278,1960.335
BC00334=752.940,3214.278,1960.335
BC00335=766.746,3215.828,1976.542
BC00336=1984.483,3218.041,658.883
BC00337=1984.483,2448.792,658.883
BC00338=1984.483,2448.792,658.883
BC00339=1984.483,2448.792,658.883
BC00340=1984.483,2448.792,658.883
BC00341=1984.483,2448.792,658.883
BC00342=1984.483,2448.792,658.883
BC00343=1984.483,2448.792,658.883
BC00344=1984.483,2448.792,658.883
BC00345=1984.483,2448.792,658.883
BC00346=1984.483,2448.792,658.883
BC00347=1984.483,2448.792,658.883
BC00348=1984.483,2448.792,658.883
BC00349=1984.483,2448.792,658.883
BC00350=1984.483,2448.792,658.883
BC00351=1984.483,2448.792,658.883
BC00352=1984.483,2448.792,658.883
BC00353=1984.483,2448.792,658.883
BC00354=1984.483,2448.792,658.883
BC00355=1984.483,2448.792,658.883
BC00356=1984.483,2448.792,658.883
BC00357=1984.483,2448.792,658.883
BC00358=1984.483,2448.792,658.883
BC00359=1984.483,2448.792,658.883
BC00360=1984.483,2448.792,658.883
BC00361=1984.483,2448.792,658.883
BC00362=1984.483,2020.544,658.883
BC00363=1984.483,2020.544,658.883
BC00364=1984.483,2020.544,658.883
BC00365=1984.483,2020.544,658.883
BC00366=1984.483,2020.544,658.883
BC00367=1984.483,2020.544,658.883
BC00368=1984.483,2020.544,658.883
BC00369=1984.470,2020.544,658.879
BC00370=1984.470,2020.544,658.879
BC00371=1984.470,2020.544,658.879
BC00372=1984.470,2020.544,658.879
BC00373=1984.470,2020.544,658.879
BC00374=1984.470,2020.544,658.879
BC00375=1984.470,2020.544,658.879
BC00376=1984.470,2020.544,658.879
BC00377=1984.470,2020.544,658.879
BC00378=1984.470,2020.544,658.879
BC00379=1984.470,2020.544,658.879
BC00380=1984.470,2020.538,658.877
BC00381=1391.860,3285.602,1013.728
BC00382=874.011,3770.839,1827.894
BC00383=779.962,3777.824,1999.134
BC00384=536.351,3774.159,1979.823
BC00385=1536.650,3350.624,1880.104
BC00386=2471.115,2623.215,1708.837
BC00387=2471.115,644.771,1708.837
BC00388=2471.115,644.771,371.374
BC00389=2499.895,888.831,371.374
BC00390=2499.895,888.831,371.366
BC00391=2499.895,888.831,371.366
BC00392=2499.895,888.831,371.366
BC00393=2499.895,888.831,371.366
BC00394=2499.895,888.831,371.366
BC00395=2499.895,888.831,371.366
BC00396=2499.895,888.831,371.366
BC00397=2499.895,888.825,371.363
BC00398=2499.895,888.825,371.363
BC00399=2499.895,888.825,371.363
BC00400=2499.895,888.825,371.363
BC00401=2499.895,888.825,371.363
BC00402=2499.895,888.825,371.363
BC00403=2499.895,888.825,371.363
BC00404=2499.895,888.825,371.363
BC00405=2499.895,888.825,371.363
BC00406=2499.895,888.825,371.363
BC00407=2499.895,888.825,371.363
BC00408=2499.895,648.814,371.363
BC00409=2499.895,648.814,371.363
BC00410=2499.895,648.814,371.363
BC00411=2499.895,648.814,371.363
BC00412=2499.895,648.814,371.363
BC00413=2499.895,648.814,371.363
BC00414=2499.895,648.814,371.363
BC00415=2499.895,648.814,371.363
BC00416=2499.895,648.814,371.363
BC00417=2499.895,648.814,371.363
BC00418=2499.895,648.814,371.363
BC00419=2499.895,648.814,371.363
BC00420=2499.895,648.814,371.363
BC00421=2499.895,648.814,371.363
BC00422=2499.895,648.814,371.363
BC00423=2499.895,648.814,371.363
BC00424=2499.895,972.335,371.363
BC00425=2499.895,972.335,371.363
BC00426=2499.895,972.335,371.363
BC00427=2204.921,409.519,319.294
BC00428=2204.921,409.519,319.294
BC00429=2204.921,409.519,319.294
BC00430=2204.921,409.519,319.294
BC00431=2204.921,409.519,319.294
BC00432=2204.921,409.519,319.294
BC00433=2204.921,409.519,319.294
BC00434=2493.165,409.519,1451.480
BC00435=2493.165,3204.728,1451.480
BC00436=430.297,4179.635,1999.619
///POSTYPE PULSE
///PULSE
EC00000=0,-1
EC00001=-811452,-554689
EC00002=-811452,-554689
EC00003=-811452,-554689
EC00004=-811452,-554689
EC00005=-811452,-554689
EC00006=-811452,-554689
EC00007=-811452,-554689
EC00008=-811450,-554689
EC00009=-811450,-554689
EC00010=-811450,-554689
EC00011=-811450,-554689
EC00012=-811450,-554689
EC00013=-811450,-554689
EC00014=-811450,-554689
EC00015=-811450,-554689
EC00016=-811450,-554689
EC00017=-811450,-554689
EC00018=-811450,-554689
EC00019=-811450,-554689
EC00020=-811450,-554689
EC00021=-811450,-554689
EC00022=-811450,-554689
EC00023=-811450,-554689
EC00024=-811450,-554689
EC00025=-811450,-554689
EC00026=-811450,-554689
EC00027=-811450,-554689
EC00028=-811450,-554689
EC00029=-811450,-554689
EC00030=-811450,-554689
EC00031=-811450,-554689
EC00032=-811450,-554689
EC00033=-811450,-554689
EC00034=-811450,-554689
EC00035=-811450,-554689
EC00036=-811450,-554689
EC00037=-811450,-554689
EC00038=-811450,-554689
EC00039=-811450,-554689
EC00040=-811450,-554689
EC00041=-811450,-554689
EC00042=-811450,-554689
EC00043=-811450,-554689
EC00044=-811450,-554689
EC00045=-811450,-554689
EC00046=-811450,-554689
EC00047=-811450,-554689
EC00048=-811450,-554689
EC00049=-811450,-554689
EC00050=-811450,-554689
EC00051=-811450,-554689
EC00052=-811450,-554689
EC00053=-811450,-554689
EC00054=-811450,-554689
EC00055=-811450,-554689
EC00056=-811450,-554689
EC00057=-811450,-554689
EC00058=-811450,-554689
EC00059=-811450,-554689
EC00060=-811450,-554689
EC00061=-811450,-554689
EC00062=-811450,-554689
EC00063=-811450,-554689
EC00064=-811450,-554689
EC00065=-811450,-554689
EC00066=-811450,-554689
EC00067=-811450,-554689
EC00068=-811450,-554689
EC00069=-811450,-554689
EC00070=-811450,-554689
EC00071=-811450,-554689
EC00072=-811450,-554689
EC00073=-811450,-554689
EC00074=-811450,-554689
EC00075=-811450,-554689
EC00076=-811450,-554689
EC00077=-811450,-554689
EC00078=-811450,-554689
EC00079=-811450,-554689
EC00080=-811450,-554689
EC00081=-811450,-554689
EC00082=-811450,-554689
EC00083=-811450,-554689
EC00084=-811450,-554689
EC00085=-811450,-554689
EC00086=-811450,-554689
EC00087=-811450,-554689
EC00088=-811450,-554689
EC00089=-811452,-554689
EC00090=-811452,-554689
EC00091=-811452,-554689
EC00092=-811452,-554689
EC00093=-811452,-554689
EC00094=-811452,-554689
EC00095=-811451,-554689
EC00096=-811451,-554689
EC00097=-811451,-554689
EC00098=-811451,-554689
EC00099=-811451,-554689
EC00100=-811451,-554689
EC00101=-811451,-554689
EC00102=-811451,-554689
EC00103=-811451,-554689
EC00104=-811451,-554689
EC00105=-811451,-554689
EC00106=-811451,-554689
EC00107=-811451,-554689
EC00108=-811451,-554689
EC00109=-811451,-554689
EC00110=-811451,-554689
EC00111=-811451,-554689
EC00112=-811451,-554689
EC00113=-811451,-554689
EC00114=-811451,-554689
EC00115=-811451,-554689
EC00116=-811451,-554689
EC00117=-811451,-554689
EC00118=-811451,-554689
EC00119=-811451,-554689
EC00120=-811451,-554689
EC00121=-811451,-554689
EC00122=-811451,-554689
EC00123=-811451,-554689
EC00124=-811451,-554689
EC00125=-811449,-554688
EC00126=-811451,-554689
EC00127=-811451,-554689
EC00128=-811451,-554689
EC00129=-811451,-554689
EC00130=-811451,-554689
EC00131=-811451,-554689
EC00132=-811451,-554689
EC00133=-811451,-554689
EC00134=-811451,-554689
EC00135=-811451,-554689
EC00136=-811451,-554689
EC00137=-811451,-554689
EC00138=-811451,-554689
EC00139=-811451,-554689
EC00140=-811451,-554689
EC00141=-811451,-554689
EC00142=-811451,-554689
EC00143=-811451,-554689
EC00144=-811451,-554689
EC00145=-363208,-550746
EC00146=-363208,-550746
EC00147=-363208,-550746
EC00148=-363208,-550746
EC00149=-363208,-550746
EC00150=-363208,-550746
EC00151=-363208,-550746
EC00152=-363208,-550746
EC00153=-363208,-550746
EC00154=-363208,-550746
EC00155=-363208,-550746
EC00156=-363208,-550746
EC00157=-363208,-550746
EC00158=-363208,-550746
EC00159=-363208,-550746
EC00160=-363208,-550746
EC00161=-363208,-550746
EC00162=-363208,-550746
EC00163=-363208,-550746
EC00164=-363208,-550746
EC00165=-363208,-550746
EC00166=-363208,-550746
EC00167=-363208,-550746
EC00168=-363208,-550746
EC00169=-363208,-550746
EC00170=-363208,-550746
EC00171=-363208,-550746
EC00172=-363208,-550746
EC00173=-363208,-550746
EC00174=-363208,-550746
EC00175=-363208,-550746
EC00176=-363208,-550746
EC00177=-363208,-550746
EC00178=-363208,-550746
EC00179=-363208,-550746
EC00180=-363208,-550746
EC00181=-363208,-550746
EC00182=-363208,-550746
EC00183=-363208,-550746
EC00184=-363208,-550746
EC00185=-363208,-550746
EC00186=-363208,-550746
EC00187=-363208,-550746
EC00188=-363208,-550746
EC00189=-363208,-550746
EC00190=-363208,-550746
EC00191=-363208,-550746
EC00192=-363208,-550746
EC00193=-363208,-550746
EC00194=-363208,-550746
EC00195=-363208,-550746
EC00196=-363208,-550746
EC00197=-363208,-550746
EC00198=-363208,-550746
EC00199=-363208,-550746
EC00200=-363208,-550746
EC00201=-363208,-550746
EC00202=-363208,-550746
EC00203=-363208,-550746
EC00204=-363208,-550746
EC00205=-363208,-550746
EC00206=-363208,-550746
EC00207=-363208,-550746
EC00208=-363208,-550746
EC00209=-363208,-550746
EC00210=-363208,-550746
EC00211=-363208,-550746
EC00212=-363208,-550746
EC00213=-363208,-550746
EC00214=-363208,-550746
EC00215=-363208,-550746
EC00216=-363208,-550746
EC00217=-363208,-550746
EC00218=-363208,-550746
EC00219=-363208,-550746
EC00220=-363208,-550746
EC00221=-363208,-550746
EC00222=-363208,-550746
EC00223=-363208,-550746
EC00224=-363208,-550746
EC00225=-363208,-550746
EC00226=-363208,-550746
EC00227=-363208,-550746
EC00228=-363207,-550746
EC00229=-363207,-550746
EC00230=-363207,-550746
EC00231=-363207,-550746
EC00232=-363207,-550746
EC00233=-363207,-550746
EC00234=-363207,-550746
EC00235=-363207,-550746
EC00236=-363207,-550746
EC00237=-363207,-550746
EC00238=-363207,-550746
EC00239=-363207,-550746
EC00240=-363207,-550746
EC00241=-363206,-550746
EC00242=-363206,-550746
EC00243=-363206,-550746
EC00244=-363206,-550746
EC00245=-363206,-550746
EC00246=-363206,-550746
EC00247=-363206,-550746
EC00248=-363206,-550746
EC00249=-363206,-550746
EC00250=-363206,-550746
EC00251=-363206,-550746
EC00252=-363206,-550746
EC00253=-363206,-550746
EC00254=-363206,-550746
EC00255=-363206,-550746
EC00256=-363206,-550746
EC00257=-363206,-550746
EC00258=-363206,-550746
EC00259=-363206,-550746
EC00260=-363206,-550746
EC00261=-363206,-550746
EC00262=-363206,-550746
EC00263=-363206,-550746
EC00264=-363206,-550746
EC00265=-363206,-550746
EC00266=-363206,-550746
EC00267=-363206,-550746
EC00268=-363206,-550746
EC00269=0,0
EC00270=-802750,0
EC00271=-802750,0
EC00272=-802750,0
EC00273=-802750,0
EC00274=-802750,0
EC00275=-802750,0
EC00276=-802750,0
EC00277=-802750,0
EC00278=-802750,0
EC00279=-802750,0
EC00280=-802750,0
EC00281=-802750,0
EC00282=-802750,0
EC00283=-802750,0
EC00284=-802750,0
EC00285=-802750,0
EC00286=-802750,0
EC00287=-802750,0
EC00288=-802750,0
EC00289=-802750,0
EC00290=-802750,0
EC00291=-802750,0
EC00292=-802750,0
EC00293=-802750,0
EC00294=-802750,0
EC00295=-802749,0
EC00296=-802749,0
EC00297=-802749,0
EC00298=-802749,0
EC00299=-802749,0
EC00300=-802749,0
EC00301=-802749,0
EC00302=-802749,0
EC00303=-802749,0
EC00304=-802749,0
EC00305=-802749,0
EC00306=-802748,0
EC00307=-802748,0
EC00308=793507,0
EC00309=793506,-1
EC00310=793506,-1
EC00311=793506,-1
EC00312=793506,-1
EC00313=793506,-1
EC00314=793506,-1
EC00315=793506,-1
EC00316=793505,-1
EC00317=793505,-1
EC00318=793505,-1
EC00319=793505,-1
EC00320=793505,-1
EC00321=793504,-1
EC00322=793504,-1
EC00323=793504,-1
EC00324=793504,-1
EC00325=793504,-1
EC00326=793504,-1
EC00327=793504,-1
EC00328=793504,-1
EC00329=793504,-1
EC00330=793504,-1
EC00331=793504,-1
EC00332=793504,-1
EC00333=793504,-1
EC00334=793504,-1
EC00335=793504,-1
EC00336=793504,-1
EC00337=793504,-1
EC00338=793504,-1
EC00339=793504,-1
EC00340=793504,-1
EC00341=793504,-1
EC00342=793504,-1
EC00343=793504,-1
EC00344=793504,-1
EC00345=793504,-1
EC00346=793504,-1
EC00347=793504,-1
EC00348=793504,-1
EC00349=793504,-1
EC00350=793504,-1
EC00351=793504,-1
EC00352=0,-1
///POSTYPE BASE
///RECTAN
///RCONF 0,0,0,0,1,0,0,0,0,0,0,0,0,0,0,0,0,0,0,0,0,0,0,0
P00006=2.006,1.622,-0.565,0.0000,0.0000,0.0000
P00021=0.073,2.058,-0.109,0.0000,0.0000,0.0000
P00022=2.006,1.622,-0.565,0.0000,0.0000,0.0000
///RCONF 0,0,0,0,0,0,0,0,0,0,0,0,0,0,0,0,0,0,0,0,0,0,0,0
P00023=-2.957,-4.083,2.762,0.0000,0.0000,0.0000
P00024=-1.466,-0.226,-0.419,0.0000,0.0000,0.0000
P00025=3.643,0.007,-2.585,0.0000,0.0000,0.0000
P00026=2.644,0.055,-2.583,0.0000,0.0000,0.0000
P00027=2.278,0.099,-4.210,0.0000,0.0000,0.0000
P00028=-1.778,-0.182,-2.050,0.0000,0.0000,0.0000
P00029=1.749,4.006,-0.261,0.0000,0.0000,0.0000
P00030=-0.014,-0.768,0.131,0.0000,0.0000,0.0000
P00031=-0.170,0.039,-0.647,0.0000,0.0000,0.0000
P00032=-0.423,0.157,3.222,0.0000,0.0000,0.0000
P00033=0.854,-1.099,3.047,0.0000,0.0000,0.0000
///RCONF 0,0,0,0,1,0,0,0,0,0,0,0,0,0,0,0,0,0,0,0,0,0,0,0
P00034=-8.151,9.743,-4.393,0.0000,0.0000,0.0000
///RCONF 0,0,0,0,0,0,0,0,0,0,0,0,0,0,0,0,0,0,0,0,0,0,0,0
P00035=0.390,-0.027,1.040,0.0000,0.0000,0.0000
P00036=-2.434,0.084,0.197,0.0000,0.0000,0.0000
P00037=-1.075,5.090,-3.949,0.0000,0.0000,0.0000
P00125=0.000,0.000,2.400,0.0000,0.0000,0.0000
///POSTYPE PULSE
///PULSE
EX00001=-798156,-1296783
//INST
///DATE 2023/12/19 17:52
///ATTR SC,RW,RJ
////FRAME ROBOT
///GROUP1 RB1,BS1
///GROUP2 ST1
NOP
SFTOF
MOVJ C00000 BC00000 VJ=100.00  +MOVJ EC00000 VJ=100.00
CALL JOB:CLEAN-R1_LONG
SFTOF
MOVJ C00001 BC00001 VJ=100.00  +MOVJ EC00001 VJ=100.00
MOVJ C00002 BC00002 VJ=100.00  +MOVJ EC00002 VJ=100.00
MOVJ C00003 BC00003 VJ=100.00  +MOVJ EC00003 VJ=100.00
'SZUKANIE
MOVJ C00004 BC00004 VJ=15.00  +MOVJ EC00004 VJ=100.00
MOVL C00005 BC00005 V=83.3  +MOVJ EC00005 VJ=15.00
REFP 3 RB1 C00006 BC00006
CALL JOB:SEARCH-R1
SET P021 P006
SFTON P021
MOVL C00007 BC00007 V=83.3  +MOVJ EC00006 VJ=15.00
REFP 3 RB1 C00008 BC00008
CALL JOB:SEARCH-R1
SET P021 P006
MOVL C00009 BC00009 V=83.3  +MOVJ EC00007 VJ=15.00
SFTOF
MOVL C00010 BC00010 V=83.3  +MOVJ EC00008 VJ=15.00
MOVL C00011 BC00011 V=83.3  +MOVJ EC00009 VJ=15.00
REFP 3 RB1 C00012 BC00012
CALL JOB:SEARCH-R1
SET P022 P006
SFTON P022
MOVL C00013 BC00013 V=83.3  +MOVJ EC00010 VJ=15.00
REFP 3 RB1 C00014 BC00014
CALL JOB:SEARCH-R1
SET P022 P006
PAUSE
SETE P022 (3) 0
PAUSE
MOVL C00015 BC00015 V=83.3  +MOVJ EC00011 VJ=15.00
SFTOF
MOVL C00016 BC00016 V=83.3  +MOVJ EC00012 VJ=15.00
MOVL C00017 BC00017 V=83.3  +MOVJ EC00013 VJ=15.00
REFP 3 RB1 C00018 BC00018
CALL JOB:SEARCH-R1
SET P023 P006
SFTON P023
MOVL C00019 BC00019 V=83.3  +MOVJ EC00014 VJ=15.00
REFP 3 RB1 C00020 BC00020
CALL JOB:SEARCH-R1
SET P023 P006
MOVL C00021 BC00021 V=83.3  +MOVJ EC00015 VJ=15.00
SFTOF
MOVL C00022 BC00022 V=83.3  +MOVJ EC00016 VJ=15.00
MOVL C00023 BC00023 V=83.3  +MOVJ EC00017 VJ=15.00
REFP 3 RB1 C00024 BC00024
CALL JOB:SEARCH-R1
SET P024 P006
SFTON P024
MOVL C00025 BC00025 V=83.3  +MOVJ EC00018 VJ=15.00
REFP 3 RB1 C00026 BC00026
CALL JOB:SEARCH-R1
SET P024 P006
MOVL C00027 BC00027 V=83.3  +MOVJ EC00019 VJ=15.00
SFTOF
MOVL C00028 BC00028 V=83.3  +MOVJ EC00020 VJ=15.00
MOVL C00029 BC00029 V=83.3  +MOVJ EC00021 VJ=15.00
REFP 3 RB1 C00030 BC00030
CALL JOB:SEARCH-R1
SET P025 P006
SFTON P025
MOVL C00031 BC00031 V=83.3  +MOVJ EC00022 VJ=15.00
REFP 3 RB1 C00032 BC00032
CALL JOB:SEARCH-R1
SET P025 P006
MOVL C00033 BC00033 V=83.3  +MOVJ EC00023 VJ=15.00
SFTOF
MOVL C00034 BC00034 V=83.3  +MOVJ EC00024 VJ=15.00
MOVL C00035 BC00035 V=83.3  +MOVJ EC00025 VJ=15.00
REFP 3 RB1 C00036 BC00036
CALL JOB:SEARCH-R1
SET P026 P006
SFTON P026
MOVL C00037 BC00037 V=83.3  +MOVJ EC00026 VJ=15.00
REFP 3 RB1 C00038 BC00038
CALL JOB:SEARCH-R1
SET P026 P006
MOVL C00039 BC00039 V=83.3  +MOVJ EC00027 VJ=15.00
SFTOF
MOVL C00040 BC00040 V=83.3  +MOVJ EC00028 VJ=15.00
MOVL C00041 BC00041 V=83.3  +MOVJ EC00029 VJ=15.00
MOVL C00042 BC00042 V=83.3  +MOVJ EC00030 VJ=15.00
REFP 3 RB1 C00043 BC00043
CALL JOB:SEARCH-R1
SET P027 P006
SFTON P027
MOVL C00044 BC00044 V=83.3  +MOVJ EC00031 VJ=15.00
REFP 3 RB1 C00045 BC00045
CALL JOB:SEARCH-R1
SET P027 P006
MOVL C00046 BC00046 V=83.3  +MOVJ EC00032 VJ=15.00
SFTOF
MOVL C00047 BC00047 V=83.3  +MOVJ EC00033 VJ=15.00
MOVL C00048 BC00048 V=83.3  +MOVJ EC00034 VJ=15.00
REFP 3 RB1 C00049 BC00049
CALL JOB:SEARCH-R1
SET P028 P006
SFTON P028
MOVL C00050 BC00050 V=83.3  +MOVJ EC00035 VJ=15.00
REFP 3 RB1 C00051 BC00051
CALL JOB:SEARCH-R1
SET P028 P006
MOVL C00052 BC00052 V=83.3  +MOVJ EC00036 VJ=15.00
SFTOF
MOVL C00053 BC00053 V=83.3  +MOVJ EC00037 VJ=15.00
MOVL C00054 BC00054 V=83.3  +MOVJ EC00038 VJ=15.00
MOVL C00055 BC00055 V=83.3  +MOVJ EC00039 VJ=15.00
REFP 3 RB1 C00056 BC00056
CALL JOB:SEARCH-R1
SET P029 P006
SFTON P029
MOVL C00057 BC00057 V=83.3  +MOVJ EC00040 VJ=15.00
REFP 3 RB1 C00058 BC00058
CALL JOB:SEARCH-R1
SET P029 P006
MOVL C00059 BC00059 V=83.3  +MOVJ EC00041 VJ=15.00
SFTOF
MOVL C00060 BC00060 V=83.3  +MOVJ EC00042 VJ=15.00
MOVL C00061 BC00061 V=83.3  +MOVJ EC00043 VJ=15.00
MOVL C00062 BC00062 V=83.3  +MOVJ EC00044 VJ=15.00
REFP 3 RB1 C00063 BC00063
CALL JOB:SEARCH-R1
SET P030 P006
SFTON P030
MOVL C00064 BC00064 V=83.3  +MOVJ EC00045 VJ=15.00
REFP 3 RB1 C00065 BC00065
CALL JOB:SEARCH-R1
SET P030 P006
MOVL C00066 BC00066 V=83.3  +MOVJ EC00046 VJ=15.00
SFTOF
MOVL C00067 BC00067 V=83.3  +MOVJ EC00047 VJ=15.00
MOVL C00068 BC00068 V=83.3  +MOVJ EC00048 VJ=15.00
REFP 3 RB1 C00069 BC00069
CALL JOB:SEARCH-R1
SET P031 P006
GETE D050 P031 (3)
SFTON P031
MOVL C00070 BC00070 V=83.3  +MOVJ EC00049 VJ=15.00
REFP 3 RB1 C00071 BC00071
CALL JOB:SEARCH-R1
SET P031 P006
SETE P031 (3) D050
MOVL C00072 BC00072 V=83.3  +MOVJ EC00050 VJ=15.00
SFTOF
MOVL C00073 BC00073 V=83.3  +MOVJ EC00051 VJ=15.00
MOVL C00074 BC00074 V=83.3  +MOVJ EC00052 VJ=15.00
REFP 3 RB1 C00075 BC00075
CALL JOB:SEARCH-R1
SET P032 P006
SFTON P032
MOVL C00076 BC00076 V=83.3  +MOVJ EC00053 VJ=15.00
REFP 3 RB1 C00077 BC00077
CALL JOB:SEARCH-R1
SET P032 P006
MOVL C00078 BC00078 V=83.3  +MOVJ EC00054 VJ=15.00
SFTOF
MOVL C00079 BC00079 V=83.3  +MOVJ EC00055 VJ=15.00
MOVL C00080 BC00080 V=83.3  +MOVJ EC00056 VJ=15.00
REFP 3 RB1 C00081 BC00081
CALL JOB:SEARCH-R1
SET P033 P006
SFTON P033
MOVL C00082 BC00082 V=83.3  +MOVJ EC00057 VJ=15.00
REFP 3 RB1 C00083 BC00083
CALL JOB:SEARCH-R1
SET P033 P006
MOVL C00084 BC00084 V=83.3  +MOVJ EC00058 VJ=15.00
SFTOF
MOVL C00085 BC00085 V=83.3  +MOVJ EC00059 VJ=15.00
MOVL C00086 BC00086 V=83.3  +MOVJ EC00060 VJ=15.00
REFP 3 RB1 C00087 BC00087
CALL JOB:SEARCH-R1
SET P034 P006
SFTON P034
MOVL C00088 BC00088 V=83.3  +MOVJ EC00061 VJ=15.00
REFP 3 RB1 C00089 BC00089
CALL JOB:SEARCH-R1
SET P034 P006
MOVL C00090 BC00090 V=83.3  +MOVJ EC00062 VJ=15.00
SFTOF
MOVL C00091 BC00091 V=83.3  +MOVJ EC00063 VJ=15.00
MOVL C00092 BC00092 V=83.3  +MOVJ EC00064 VJ=15.00
REFP 3 RB1 C00093 BC00093
CALL JOB:SEARCH-R1
SET P035 P006
SFTON P035
MOVL C00094 BC00094 V=83.3  +MOVJ EC00065 VJ=15.00
REFP 3 RB1 C00095 BC00095
CALL JOB:SEARCH-R1
SET P035 P006
MOVL C00096 BC00096 V=83.3  +MOVJ EC00066 VJ=15.00
SFTOF
MOVL C00097 BC00097 V=83.3  +MOVJ EC00067 VJ=15.00
MOVL C00098 BC00098 V=83.3  +MOVJ EC00068 VJ=15.00
REFP 3 RB1 C00099 BC00099
CALL JOB:SEARCH-R1
SET P036 P006
SFTON P036
MOVL C00100 BC00100 V=83.3  +MOVJ EC00069 VJ=15.00
REFP 3 RB1 C00101 BC00101
CALL JOB:SEARCH-R1
SET P036 P006
MOVL C00102 BC00102 V=83.3  +MOVJ EC00070 VJ=15.00
SFTOF
MOVL C00103 BC00103 V=83.3  +MOVJ EC00071 VJ=15.00
MOVJ C00104 BC00104 VJ=100.00  +MOVJ EC00072 VJ=15.00
MOVJ C00105 BC00105 VJ=100.00  +MOVJ EC00073 VJ=100.00
MOVJ C00106 BC00106 VJ=100.00  +MOVJ EC00074 VJ=100.00
MOVL C00107 BC00107 V=83.3  +MOVJ EC00075 VJ=15.00
REFP 3 RB1 C00108 BC00108
CALL JOB:SEARCH-R1
SET P037 P006
SFTON P037
MOVL C00109 BC00109 V=83.3  +MOVJ EC00076 VJ=15.00
REFP 3 RB1 C00110 BC00110
CALL JOB:SEARCH-R1
SET P037 P006
MOVL C00111 BC00111 V=83.3  +MOVJ EC00077 VJ=15.00
SFTOF
MOVL C00112 BC00112 V=166.7  +MOVJ EC00078 VJ=15.00
SFTON P037
MACRO1 MJ#(0) ARGF7
MOVL C00113 BC00113 V=83.3  +MOVJ EC00079 VJ=100.00
ARCON
MOVL C00114 BC00114 V=10.0  +MOVJ EC00080 VJ=100.00
MOVL C00115 BC00115 V=10.0  +MOVJ EC00081 VJ=100.00
MOVL C00116 BC00116 V=10.0  +MOVJ EC00082 VJ=100.00
MOVL C00117 BC00117 V=10.0  +MOVJ EC00083 VJ=100.00
MOVL C00118 BC00118 V=10.0  +MOVJ EC00084 VJ=100.00
MOVL C00119 BC00119 V=10.0  +MOVJ EC00085 VJ=100.00
MOVL C00120 BC00120 V=10.0  +MOVJ EC00086 VJ=100.00
SFTON P021
ARCON
MOVL C00121 BC00121 V=10.0  +MOVJ EC00087 VJ=100.00
MOVL C00122 BC00122 V=10.0  +MOVJ EC00088 VJ=100.00
MOVL C00123 BC00123 V=10.0  +MOVJ EC00089 VJ=100.00
MOVL C00124 BC00124 V=10.0  +MOVJ EC00090 VJ=20.00
SFTON P022
MOVL C00125 BC00125 V=10.0  +MOVJ EC00091 VJ=20.00
SFTON P023
MOVL C00126 BC00126 V=10.0  +MOVJ EC00092 VJ=20.00
SFTON P024
MOVL C00127 BC00127 V=10.0  +MOVJ EC00093 VJ=20.00
MOVL C00128 BC00128 V=10.0  +MOVJ EC00094 VJ=20.00
ARCOF
MOVJ C00129 BC00129 VJ=20.00  +MOVJ EC00095 VJ=20.00
SFTOF
MOVJ C00130 BC00130 VJ=100.00  +MOVJ EC00096 VJ=20.00
MOVJ C00131 BC00131 VJ=100.00  +MOVJ EC00097 VJ=20.00
SFTON P036
MOVJ C00132 BC00132 VJ=20.00  +MOVJ EC00098 VJ=100.00
ARCON
MOVL C00133 BC00133 V=10.0  +MOVJ EC00099 VJ=20.00
MOVL C00134 BC00134 V=10.0  +MOVJ EC00100 VJ=20.00
MOVL C00135 BC00135 V=10.0  +MOVJ EC00101 VJ=20.00
MOVL C00136 BC00136 V=10.0  +MOVJ EC00102 VJ=20.00
MOVL C00137 BC00137 V=10.0  +MOVJ EC00103 VJ=20.00
MOVL C00138 BC00138 V=10.0  +MOVJ EC00104 VJ=20.00
MOVL C00139 BC00139 V=10.0  +MOVJ EC00105 VJ=20.00
MOVL C00140 BC00140 V=10.0  +MOVJ EC00106 VJ=20.00
MOVL C00141 BC00141 V=10.0  +MOVJ EC00107 VJ=20.00
SFTON P035
MOVL C00142 BC00142 V=10.0  +MOVJ EC00108 VJ=20.00
MOVL C00143 BC00143 V=10.0  +MOVJ EC00109 VJ=15.00
SFTON P034
MOVL C00144 BC00144 V=10.0  +MOVJ EC00110 VJ=15.00
SFTON P033
MOVL C00145 BC00145 V=10.0  +MOVJ EC00111 VJ=15.00
SFTON P032
MOVL C00146 BC00146 V=10.0  +MOVJ EC00112 VJ=15.00
MOVL C00147 BC00147 V=10.0  +MOVJ EC00113 VJ=15.00
ARCOF
MOVJ C00148 BC00148 VJ=15.00  +MOVJ EC00114 VJ=15.00
SFTOF
MOVJ C00149 BC00149 VJ=100.00  +MOVJ EC00115 VJ=20.00
SFTON P028
MOVJ C00150 BC00150 VJ=20.00  +MOVJ EC00116 VJ=20.00
ARCON
MOVL C00151 BC00151 V=8.3  +MOVJ EC00117 VJ=20.00
SFTON P027
MOVL C00152 BC00152 V=10.0  +MOVJ EC00118 VJ=20.00
MOVL C00153 BC00153 V=10.0  +MOVJ EC00119 VJ=20.00
MOVL C00154 BC00154 V=10.0  +MOVJ EC00120 VJ=100.00
MOVL C00155 BC00155 V=10.0  +MOVJ EC00121 VJ=20.00
SFTON P026
MOVL C00156 BC00156 V=10.0  +MOVJ EC00122 VJ=20.00
MOVL C00157 BC00157 V=10.0  +MOVJ EC00123 VJ=20.00
MOVL C00158 BC00158 V=10.8  +MOVJ EC00124 VJ=20.00
MOVL C00159 BC00159 V=10.8  +MOVJ EC00125 VJ=20.00
SFTON P025
MOVL C00160 BC00160 V=10.8  +MOVJ EC00126 VJ=20.00
MOVL C00161 BC00161 V=10.8  +MOVJ EC00127 VJ=20.00
ARCOF
MOVJ C00162 BC00162 VJ=20.00  +MOVJ EC00128 VJ=20.00
SFTOF
MOVJ C00163 BC00163 VJ=100.00  +MOVJ EC00129 VJ=20.00
MOVJ C00164 BC00164 VJ=100.00  +MOVJ EC00130 VJ=20.00
SFTON P028
MOVJ C00165 BC00165 VJ=20.00  +MOVJ EC00131 VJ=20.00
ARCON
MOVL C00166 BC00166 V=10.0  +MOVJ EC00132 VJ=20.00
SFTON P029
MOVL C00167 BC00167 V=10.0  +MOVJ EC00133 VJ=20.00
MOVL C00168 BC00168 V=10.0  +MOVJ EC00134 VJ=20.00
MOVL C00169 BC00169 V=10.0  +MOVJ EC00135 VJ=20.00
MOVL C00170 BC00170 V=10.0  +MOVJ EC00136 VJ=20.00
SFTON P030
MOVL C00171 BC00171 V=10.0  +MOVJ EC00137 VJ=20.00
MOVL C00172 BC00172 V=10.0  +MOVJ EC00138 VJ=20.00
MOVL C00173 BC00173 V=10.0  +MOVJ EC00139 VJ=20.00
MOVL C00174 BC00174 V=10.0  +MOVJ EC00140 VJ=20.00
SFTON P031
MOVL C00175 BC00175 V=10.0  +MOVJ EC00141 VJ=20.00
MOVL C00176 BC00176 V=10.0  +MOVJ EC00142 VJ=20.00
ARCOF
MOVJ C00177 BC00177 VJ=20.00  +MOVJ EC00143 VJ=20.00
SFTOF
MOVJ C00178 BC00178 VJ=100.00  +MOVJ EC00144 VJ=100.00
MOVJ C00179 BC00179 VJ=100.00  +MOVJ EC00145 VJ=100.00
CALL JOB:CLEAN-R1_LONG
MOVJ C00180 BC00180 VJ=100.00  +MOVJ EC00146 VJ=100.00
MOVJ C00181 BC00181 VJ=100.00  +MOVJ EC00147 VJ=100.00
PAUSE
'SZUKANIE DRUGA STRONA
MOVJ C00182 BC00182 VJ=15.00  +MOVJ EC00148 VJ=15.00
SFTOF
MOVL C00183 BC00183 V=83.3  +MOVJ EC00149 VJ=15.00
REFP 3 RB1 C00184 BC00184
CALL JOB:SEARCH-R1
SET P035 P006
SFTON P035
MOVL C00185 BC00185 V=83.3  +MOVJ EC00150 VJ=15.00
REFP 3 RB1 C00186 BC00186
CALL JOB:SEARCH-R1
SET P035 P006
MOVL C00187 BC00187 V=83.3  +MOVJ EC00151 VJ=15.00
SFTOF
MOVL C00188 BC00188 V=166.7  +MOVJ EC00152 VJ=15.00
MOVL C00189 BC00189 V=83.3  +MOVJ EC00153 VJ=15.00
REFP 3 RB1 C00190 BC00190
CALL JOB:SEARCH-R1
SET P021 P006
SFTON P021
MOVL C00191 BC00191 V=83.3  +MOVJ EC00154 VJ=15.00
REFP 3 RB1 C00192 BC00192
CALL JOB:SEARCH-R1
SET P021 P006
MOVL C00193 BC00193 V=83.3  +MOVJ EC00155 VJ=15.00
SFTOF
MOVL C00194 BC00194 V=83.3  +MOVJ EC00156 VJ=100.00
SFTOF
MOVL C00195 BC00195 V=83.3  +MOVJ EC00157 VJ=15.00
REFP 3 RB1 C00196 BC00196
CALL JOB:SEARCH-R1
SET P022 P006
SFTON P022
MOVL C00197 BC00197 V=83.3  +MOVJ EC00158 VJ=15.00
REFP 3 RB1 C00198 BC00198
CALL JOB:SEARCH-R1
SET P022 P006
MOVL C00199 BC00199 V=83.3  +MOVJ EC00159 VJ=15.00
SFTOF
MOVL C00200 BC00200 V=83.3  +MOVJ EC00160 VJ=15.00
MOVL C00201 BC00201 V=83.3  +MOVJ EC00161 VJ=15.00
REFP 3 RB1 C00202 BC00202
CALL JOB:SEARCH-R1
SET P023 P006
SFTON P023
MOVL C00203 BC00203 V=83.3  +MOVJ EC00162 VJ=15.00
REFP 3 RB1 C00204 BC00204
CALL JOB:SEARCH-R1
SET P023 P006
MOVL C00205 BC00205 V=83.3  +MOVJ EC00163 VJ=15.00
SFTOF
MOVL C00206 BC00206 V=83.3  +MOVJ EC00164 VJ=15.00
MOVL C00207 BC00207 V=83.3  +MOVJ EC00165 VJ=15.00
REFP 3 RB1 C00208 BC00208
CALL JOB:SEARCH-R1
SET P024 P006
SFTON P024
MOVL C00209 BC00209 V=83.3  +MOVJ EC00166 VJ=15.00
REFP 3 RB1 C00210 BC00210
CALL JOB:SEARCH-R1
SET P024 P006
MOVL C00211 BC00211 V=83.3  +MOVJ EC00167 VJ=15.00
SFTOF
MOVJ C00212 BC00212 VJ=15.00  +MOVJ EC00168 VJ=0.78
MOVJ C00213 BC00213 VJ=15.00  +MOVJ EC00169 VJ=15.00
MOVL C00214 BC00214 V=83.3  +MOVJ EC00170 VJ=15.00
REFP 3 RB1 C00215 BC00215
CALL JOB:SEARCH-R1
SET P025 P006
SFTON P025
MOVL C00216 BC00216 V=83.3  +MOVJ EC00171 VJ=15.00
REFP 3 RB1 C00217 BC00217
CALL JOB:SEARCH-R1
SET P025 P006
MOVL C00218 BC00218 V=83.3  +MOVJ EC00172 VJ=15.00
SFTOF
MOVL C00219 BC00219 V=83.3  +MOVJ EC00173 VJ=15.00
MOVL C00220 BC00220 V=83.3  +MOVJ EC00174 VJ=15.00
REFP 3 RB1 C00221 BC00221
CALL JOB:SEARCH-R1
SET P026 P006
SFTON P026
MOVL C00222 BC00222 V=83.3  +MOVJ EC00175 VJ=15.00
REFP 3 RB1 C00223 BC00223
CALL JOB:SEARCH-R1
SET P026 P006
MOVL C00224 BC00224 V=83.3  +MOVJ EC00176 VJ=15.00
SFTOF
MOVL C00225 BC00225 V=83.3  +MOVJ EC00177 VJ=15.00
MOVL C00226 BC00226 V=83.3  +MOVJ EC00178 VJ=15.00
REFP 3 RB1 C00227 BC00227
CALL JOB:SEARCH-R1
SET P027 P006
SFTON P027
MOVL C00228 BC00228 V=83.3  +MOVJ EC00179 VJ=15.00
REFP 3 RB1 C00229 BC00229
CALL JOB:SEARCH-R1
SET P027 P006
MOVL C00230 BC00230 V=83.3  +MOVJ EC00180 VJ=15.00
SFTOF
MOVL C00231 BC00231 V=83.3  +MOVJ EC00181 VJ=15.00
MOVL C00232 BC00232 V=83.3  +MOVJ EC00182 VJ=15.00
REFP 3 RB1 C00233 BC00233
CALL JOB:SEARCH-R1
SET P028 P006
SFTON P028
MOVL C00234 BC00234 V=83.3  +MOVJ EC00183 VJ=15.00
REFP 3 RB1 C00235 BC00235
CALL JOB:SEARCH-R1
SET P028 P006
MOVL C00236 BC00236 V=83.3  +MOVJ EC00184 VJ=15.00
SFTOF
MOVL C00237 BC00237 V=83.3  +MOVJ EC00185 VJ=15.00
MOVL C00238 BC00238 V=83.3  +MOVJ EC00186 VJ=15.00
REFP 3 RB1 C00239 BC00239
CALL JOB:SEARCH-R1
SET P029 P006
SFTON P029
MOVL C00240 BC00240 V=83.3  +MOVJ EC00187 VJ=15.00
REFP 3 RB1 C00241 BC00241
CALL JOB:SEARCH-R1
SET P029 P006
MOVL C00242 BC00242 V=83.3  +MOVJ EC00188 VJ=15.00
SFTOF
MOVJ C00243 BC00243 VJ=15.00  +MOVJ EC00189 VJ=15.00
MOVJ C00244 BC00244 VJ=15.00  +MOVJ EC00190 VJ=15.00
MOVL C00245 BC00245 V=83.3  +MOVJ EC00191 VJ=15.00
REFP 3 RB1 C00246 BC00246
CALL JOB:SEARCH-R1
SET P030 P006
SFTON P030
MOVL C00247 BC00247 V=83.3  +MOVJ EC00192 VJ=15.00
REFP 3 RB1 C00248 BC00248
CALL JOB:SEARCH-R1
SET P030 P006
MOVL C00249 BC00249 V=83.3  +MOVJ EC00193 VJ=15.00
SFTOF
MOVL C00250 BC00250 V=83.3  +MOVJ EC00194 VJ=15.00
MOVL C00251 BC00251 V=83.3  +MOVJ EC00195 VJ=15.00
REFP 3 RB1 C00252 BC00252
CALL JOB:SEARCH-R1
SET P031 P006
MOVL C00253 BC00253 V=83.3  +MOVJ EC00196 VJ=15.00
REFP 3 RB1 C00254 BC00254
CALL JOB:SEARCH-R1
SET P031 P006
MOVL C00255 BC00255 V=83.3  +MOVJ EC00197 VJ=15.00
SFTOF
MOVL C00256 BC00256 V=83.3  +MOVJ EC00198 VJ=15.00
MOVL C00257 BC00257 V=83.3  +MOVJ EC00199 VJ=15.00
MOVL C00258 BC00258 V=16.7 SRCH RIN#(1)=ON DIS=20.0  +MOVJ EC00200 VJ=0.78
IMOV P125 V=23.0  +IMOV EX001
PAUSE
REFP 3 RB1 C00259 BC00259
CALL JOB:SEARCH-R1
SET P032 P006
GETE D050 P032 (3)
MOVL C00260 BC00260 V=83.3  +MOVJ EC00201 VJ=15.00
REFP 3 RB1 C00261 BC00261
CALL JOB:SEARCH-R1
SET P032 P006
SETE P032 (3) D050
MOVL C00262 BC00262 V=83.3  +MOVJ EC00202 VJ=15.00
SFTOF
MOVL C00263 BC00263 V=250.0  +MOVJ EC00203 VJ=15.00
MOVL C00264 BC00264 V=83.3  +MOVJ EC00204 VJ=15.00
REFP 3 RB1 C00265 BC00265
CALL JOB:SEARCH-R1
SET P033 P006
SFTON P033
MOVL C00266 BC00266 V=83.3  +MOVJ EC00205 VJ=15.00
REFP 3 RB1 C00267 BC00267
CALL JOB:SEARCH-R1
SET P033 P006
MOVL C00268 BC00268 V=83.3  +MOVJ EC00206 VJ=15.00
SFTOF
MOVJ C00269 BC00269 VJ=15.00  +MOVJ EC00207 VJ=15.00
MOVL C00270 BC00270 V=83.3  +MOVJ EC00208 VJ=15.00
REFP 3 RB1 C00271 BC00271
CALL JOB:SEARCH-R1
SET P034 P006
SFTON P034
MOVL C00272 BC00272 V=83.3  +MOVJ EC00209 VJ=15.00
REFP 3 RB1 C00273 BC00273
CALL JOB:SEARCH-R1
SET P034 P006
MOVL C00274 BC00274 V=83.3  +MOVJ EC00210 VJ=15.00
MOVJ C00275 BC00275 VJ=15.00  +MOVJ EC00211 VJ=15.00
'KONIEC SZUKANIE DRUGA STRONA
'SPAWANIE DRUGA STRONA
MOVJ C00276 BC00276 VJ=15.00  +MOVJ EC00212 VJ=15.00
MACRO1 MJ#(0) ARGF7
SFTOF
SFTON P034
MOVJ C00277 BC00277 VJ=15.00  +MOVJ EC00213 VJ=15.00
ARCON
MOVL C00278 BC00278 V=10.0  +MOVJ EC00214 VJ=15.00
MOVL C00279 BC00279 V=10.0  +MOVJ EC00215 VJ=15.00
SFTOF
SFTON P033
MOVL C00280 BC00280 V=10.0  +MOVJ EC00216 VJ=15.00
MOVL C00281 BC00281 V=10.0  +MOVJ EC00217 VJ=15.00
SFTOF
PAUSE
SFTON P032
MOVL C00282 BC00282 V=10.0  +MOVJ EC00218 VJ=15.00
SFTOF
SFTON P031
MOVL C00283 BC00283 V=10.0  +MOVJ EC00219 VJ=15.00
SFTOF
SFTON P030
MOVL C00284 BC00284 V=10.0  +MOVJ EC00220 VJ=15.00
MOVL C00285 BC00285 V=10.0  +MOVJ EC00221 VJ=15.00
MOVL C00286 BC00286 V=10.0  +MOVJ EC00222 VJ=15.00
ARCOF
SFTOF
MOVJ C00287 BC00287 VJ=15.00  +MOVJ EC00223 VJ=15.00
MOVJ C00288 BC00288 VJ=50.00  +MOVJ EC00224 VJ=15.00
MOVJ C00289 BC00289 VJ=50.00  +MOVJ EC00225 VJ=50.00
MOVJ C00290 BC00290 VJ=50.00  +MOVJ EC00226 VJ=50.00
MOVJ C00291 BC00291 VJ=50.00  +MOVJ EC00227 VJ=50.00
SFTON P035
MOVL C00292 BC00292 V=83.3  +MOVJ EC00228 VJ=50.00
ARCON
MOVL C00293 BC00293 V=10.0  +MOVJ EC00229 VJ=50.00
MOVL C00294 BC00294 V=10.0  +MOVJ EC00230 VJ=50.00
SFTON P021
MOVL C00295 BC00295 V=10.0  +MOVJ EC00231 VJ=50.00
MOVL C00296 BC00296 V=10.0  +MOVJ EC00232 VJ=50.00
SFTON P022
MOVL C00297 BC00297 V=10.0  +MOVJ EC00233 VJ=50.00
SFTON P023
MOVL C00298 BC00298 V=10.0  +MOVJ EC00234 VJ=50.00
SFTON P024
MOVL C00299 BC00299 V=10.0  +MOVJ EC00235 VJ=50.00
MOVL C00300 BC00300 V=10.0  +MOVJ EC00236 VJ=50.00
MOVL C00301 BC00301 V=10.0  +MOVJ EC00237 VJ=50.00
ARCOF
MOVJ C00302 BC00302 VJ=20.00  +MOVJ EC00238 VJ=50.00
MOVJ C00303 BC00303 VJ=50.00  +MOVJ EC00239 VJ=20.00
SFTON P027
MOVJ C00304 BC00304 VJ=15.00  +MOVJ EC00240 VJ=50.00
ARCON
MOVL C00305 BC00305 V=10.0  +MOVJ EC00241 VJ=15.00
MOVL C00306 BC00306 V=10.0  +MOVJ EC00242 VJ=15.00
MOVL C00307 BC00307 V=10.0  +MOVJ EC00243 VJ=15.00
MOVL C00308 BC00308 V=10.0  +MOVJ EC00244 VJ=15.00
SFTON P028
MOVL C00309 BC00309 V=10.0  +MOVJ EC00245 VJ=15.00
MOVL C00310 BC00310 V=10.0  +MOVJ EC00246 VJ=15.00
MOVL C00311 BC00311 V=10.0  +MOVJ EC00247 VJ=15.00
MOVL C00312 BC00312 V=10.0  +MOVJ EC00248 VJ=15.00
SFTON P029
MOVL C00313 BC00313 V=10.0  +MOVJ EC00249 VJ=15.00
MOVL C00314 BC00314 V=10.0  +MOVJ EC00250 VJ=15.00
ARCOF
MOVJ C00315 BC00315 VJ=15.00  +MOVJ EC00251 VJ=15.00
MOVJ C00316 BC00316 VJ=15.00  +MOVJ EC00252 VJ=15.00
SFTOF
MOVJ C00317 BC00317 VJ=15.00  +MOVJ EC00253 VJ=15.00
SFTON P027
MOVJ C00318 BC00318 VJ=15.00  +MOVJ EC00254 VJ=15.00
ARCON
MOVL C00319 BC00319 V=10.0  +MOVJ EC00255 VJ=15.00
MOVL C00320 BC00320 V=10.0  +MOVJ EC00256 VJ=15.00
MOVL C00321 BC00321 V=10.0  +MOVJ EC00257 VJ=15.00
MOVL C00322 BC00322 V=10.0  +MOVJ EC00258 VJ=15.00
SFTON P026
MOVL C00323 BC00323 V=10.0  +MOVJ EC00259 VJ=15.00
MOVL C00324 BC00324 V=10.0  +MOVJ EC00260 VJ=15.00
MOVL C00325 BC00325 V=10.0  +MOVJ EC00261 VJ=15.00
MOVL C00326 BC00326 V=10.0  +MOVJ EC00262 VJ=15.00
SFTON P025
MOVL C00327 BC00327 V=10.0  +MOVJ EC00263 VJ=15.00
MOVL C00328 BC00328 V=10.0  +MOVJ EC00264 VJ=15.00
MOVL C00329 BC00329 V=10.0  +MOVJ EC00265 VJ=15.00
ARCOF
MOVJ C00330 BC00330 VJ=15.00  +MOVJ EC00266 VJ=15.00
SFTOF
MOVJ C00331 BC00331 VJ=100.00  +MOVJ EC00267 VJ=15.00
MOVJ C00332 BC00332 VJ=100.00  +MOVJ EC00268 VJ=100.00
MOVJ C00333 BC00333 VJ=100.00  +MOVJ EC00269 VJ=100.00
MOVJ C00334 BC00334 VJ=100.00  +MOVJ EC00270 VJ=100.00
CALL JOB:CLEAN-R1_LONG
MOVJ C00335 BC00335 VJ=100.00  +MOVJ EC00271 VJ=100.00
MOVJ C00336 BC00336 VJ=100.00  +MOVJ EC00272 VJ=100.00
MOVJ C00337 BC00337 VJ=100.00  +MOVJ EC00273 VJ=100.00
MOVL C00338 BC00338 V=83.3  +MOVJ EC00274 VJ=15.00
REFP 3 RB1 C00339 BC00339
CALL JOB:SEARCH-R1
SET P021 P006
SFTON P021
MOVL C00340 BC00340 V=83.3  +MOVJ EC00275 VJ=15.00
REFP 3 RB1 C00341 BC00341
CALL JOB:SEARCH-R1
SET P021 P006
MOVL C00342 BC00342 V=83.3  +MOVJ EC00276 VJ=15.00
SFTOF
MOVL C00343 BC00343 V=166.7  +MOVJ EC00277 VJ=15.00
MOVL C00344 BC00344 V=83.3  +MOVJ EC00278 VJ=15.00
REFP 3 RB1 C00345 BC00345
CALL JOB:SEARCH-R1
SET P022 P006
SFTON P022
MOVL C00346 BC00346 V=83.3  +MOVJ EC00279 VJ=15.00
REFP 3 RB1 C00347 BC00347
CALL JOB:SEARCH-R1
SET P022 P006
MOVL C00348 BC00348 V=83.3  +MOVJ EC00280 VJ=15.00
SFTOF
MOVL C00349 BC00349 V=166.7  +MOVJ EC00281 VJ=15.00
MOVL C00350 BC00350 V=83.3  +MOVJ EC00282 VJ=15.00
REFP 3 RB1 C00351 BC00351
CALL JOB:SEARCH-R1
SET P023 P006
SFTON P023
MOVL C00352 BC00352 V=83.3  +MOVJ EC00283 VJ=15.00
REFP 3 RB1 C00353 BC00353
CALL JOB:SEARCH-R1
SET P023 P006
MOVL C00354 BC00354 V=83.3  +MOVJ EC00284 VJ=15.00
SFTOF
MOVL C00355 BC00355 V=166.7  +MOVJ EC00285 VJ=15.00
MOVL C00356 BC00356 V=83.3  +MOVJ EC00286 VJ=15.00
REFP 3 RB1 C00357 BC00357
CALL JOB:SEARCH-R1
SET P024 P006
SFTON P024
MOVL C00358 BC00358 V=83.3  +MOVJ EC00287 VJ=15.00
REFP 3 RB1 C00359 BC00359
CALL JOB:SEARCH-R1
SET P024 P006
MOVL C00360 BC00360 V=83.3  +MOVJ EC00288 VJ=15.00
SFTOF
MOVL C00361 BC00361 V=166.7  +MOVJ EC00289 VJ=15.00
MOVL C00362 BC00362 V=83.3  +MOVJ EC00290 VJ=15.00
REFP 3 RB1 C00363 BC00363
CALL JOB:SEARCH-R1
SET P025 P006
SFTON P025
MOVL C00364 BC00364 V=83.3  +MOVJ EC00291 VJ=15.00
REFP 3 RB1 C00365 BC00365
CALL JOB:SEARCH-R1
SET P025 P006
MOVL C00366 BC00366 V=83.3  +MOVJ EC00292 VJ=15.00
SFTOF
MOVJ C00367 BC00367 VJ=30.00  +MOVJ EC00293 VJ=100.00
MOVJ C00368 BC00368 VJ=30.00  +MOVJ EC00294 VJ=30.00
SFTON P023
MACRO1 MJ#(0) ARGF7
MOVL C00369 BC00369 V=83.3  +MOVJ EC00295 VJ=30.00
ARCON
SFTON P022
MOVL C00370 BC00370 V=10.8  +MOVJ EC00296 VJ=30.00
SFTON P021
MOVL C00371 BC00371 V=10.8  +MOVJ EC00297 VJ=30.00
MOVL C00372 BC00372 V=10.8  +MOVJ EC00298 VJ=30.00
ARCOF
SFTOF
MOVJ C00373 BC00373 VJ=30.00  +MOVJ EC00299 VJ=30.00
MOVJ C00374 BC00374 VJ=30.00  +MOVJ EC00300 VJ=30.00
SFTON P023
MOVL C00375 BC00375 V=83.3  +MOVJ EC00301 VJ=30.00
ARCON
SFTON P024
MOVL C00376 BC00376 V=10.8  +MOVJ EC00302 VJ=30.00
SFTON P025
MOVL C00377 BC00377 V=10.8  +MOVJ EC00303 VJ=30.00
MOVL C00378 BC00378 V=10.8  +MOVJ EC00304 VJ=30.00
MOVL C00379 BC00379 V=10.8  +MOVJ EC00305 VJ=30.00
ARCOF
SFTOF
MOVJ C00380 BC00380 VJ=30.00  +MOVJ EC00306 VJ=30.00
MOVJ C00381 BC00381 VJ=30.00  +MOVJ EC00307 VJ=30.00
MOVJ C00382 BC00382 VJ=100.00  +MOVJ EC00308 VJ=100.00
MOVJ C00383 BC00383 VJ=30.00  +MOVJ EC00309 VJ=30.00
CALL JOB:ONLYCUT-R1_LONG
MOVJ C00384 BC00384 VJ=30.00  +MOVJ EC00310 VJ=30.00
MOVJ C00385 BC00385 VJ=100.00  +MOVJ EC00311 VJ=100.00
MOVJ C00386 BC00386 VJ=30.00  +MOVJ EC00312 VJ=30.00
MOVJ C00387 BC00387 VJ=30.00  +MOVJ EC00313 VJ=30.00
MOVJ C00388 BC00388 VJ=30.00  +MOVJ EC00314 VJ=30.00
MOVJ C00389 BC00389 VJ=30.00  +MOVJ EC00315 VJ=30.00
MOVJ C00390 BC00390 VJ=100.00  +MOVJ EC00316 VJ=100.00
MOVL C00391 BC00391 V=83.3  +MOVJ EC00317 VJ=15.00
REFP 3 RB1 C00392 BC00392
CALL JOB:SEARCH-R1
SET P021 P006
SFTON P021
MOVL C00393 BC00393 V=83.3  +MOVJ EC00318 VJ=15.00
REFP 3 RB1 C00394 BC00394
CALL JOB:SEARCH-R1
SET P021 P006
MOVL C00395 BC00395 V=83.3  +MOVJ EC00319 VJ=15.00
SFTOF
MOVL C00396 BC00396 V=166.7  +MOVJ EC00320 VJ=15.00
MOVL C00397 BC00397 V=83.3  +MOVJ EC00321 VJ=15.00
REFP 3 RB1 C00398 BC00398
CALL JOB:SEARCH-R1
SET P022 P006
SFTON P022
MOVL C00399 BC00399 V=83.3  +MOVJ EC00322 VJ=15.00
REFP 3 RB1 C00400 BC00400
CALL JOB:SEARCH-R1
SET P022 P006
MOVL C00401 BC00401 V=83.3  +MOVJ EC00323 VJ=15.00
SFTOF
MOVL C00402 BC00402 V=166.7  +MOVJ EC00324 VJ=15.00
MOVL C00403 BC00403 V=83.3  +MOVJ EC00325 VJ=15.00
REFP 3 RB1 C00404 BC00404
CALL JOB:SEARCH-R1
SET P023 P006
SFTON P023
MOVL C00405 BC00405 V=83.3  +MOVJ EC00326 VJ=15.00
REFP 3 RB1 C00406 BC00406
CALL JOB:SEARCH-R1
SET P023 P006
MOVL C00407 BC00407 V=83.3  +MOVJ EC00327 VJ=15.00
SFTOF
MOVL C00408 BC00408 V=166.7  +MOVJ EC00328 VJ=15.00
MOVL C00409 BC00409 V=83.3  +MOVJ EC00329 VJ=15.00
REFP 3 RB1 C00410 BC00410
CALL JOB:SEARCH-R1
SET P024 P006
SFTON P024
MOVL C00411 BC00411 V=83.3  +MOVJ EC00330 VJ=15.00
REFP 3 RB1 C00412 BC00412
CALL JOB:SEARCH-R1
SET P024 P006
MOVL C00413 BC00413 V=83.3  +MOVJ EC00331 VJ=15.00
SFTOF
MOVL C00414 BC00414 V=166.7  +MOVJ EC00332 VJ=15.00
MOVL C00415 BC00415 V=83.3  +MOVJ EC00333 VJ=15.00
REFP 3 RB1 C00416 BC00416
CALL JOB:SEARCH-R1
SET P025 P006
SFTON P025
MOVL C00417 BC00417 V=83.3  +MOVJ EC00334 VJ=15.00
REFP 3 RB1 C00418 BC00418
CALL JOB:SEARCH-R1
SET P025 P006
MOVL C00419 BC00419 V=83.3  +MOVJ EC00335 VJ=15.00
SFTOF
MOVJ C00420 BC00420 VJ=30.00  +MOVJ EC00336 VJ=100.00
MOVJ C00421 BC00421 VJ=30.00  +MOVJ EC00337 VJ=30.00
SFTON P023
MOVL C00422 BC00422 V=83.3  +MOVJ EC00338 VJ=30.00
ARCON
SFTON P022
MOVL C00423 BC00423 V=10.8  +MOVJ EC00339 VJ=30.00
SFTON P021
MOVL C00424 BC00424 V=10.8  +MOVJ EC00340 VJ=30.00
MOVL C00425 BC00425 V=10.8  +MOVJ EC00341 VJ=30.00
ARCOF
SFTOF
MOVJ C00426 BC00426 VJ=30.00  +MOVJ EC00342 VJ=30.00
MOVJ C00427 BC00427 VJ=30.00  +MOVJ EC00343 VJ=30.00
SFTON P023
MOVL C00428 BC00428 V=83.3  +MOVJ EC00344 VJ=30.00
ARCON
SFTON P024
MOVL C00429 BC00429 V=10.8  +MOVJ EC00345 VJ=30.00
SFTON P025
MOVL C00430 BC00430 V=10.8  +MOVJ EC00346 VJ=30.00
MOVL C00431 BC00431 V=10.8  +MOVJ EC00347 VJ=30.00
MOVL C00432 BC00432 V=10.8  +MOVJ EC00348 VJ=30.00
ARCOF
SFTOF
MOVJ C00433 BC00433 VJ=30.00  +MOVJ EC00349 VJ=30.00
MOVJ C00434 BC00434 VJ=30.00  +MOVJ EC00350 VJ=30.00
MOVJ C00435 BC00435 VJ=30.00  +MOVJ EC00351 VJ=30.00
MOVJ C00436 BC00436 VJ=30.00  +MOVJ EC00352 VJ=30.00
END
